LIN {X -117.977,Y -5.308,Z -33.189,A -90.000,B 90.000,C 0.000} C_DIS
LIN {X -117.973,Y -5.308,Z -33.170,A -90.000,B 90.000,C 0.000} C_DIS
LIN {X -117.912,Y -5.308,Z -32.912,A -90.000,B 90.000,C 0.000} C_DIS
LIN {X -117.911,Y -5.308,Z -32.907,A -90.000,B 90.000,C 0.000} C_DIS
LIN {X -117.908,Y -5.308,Z -32.898,A -90.000,B 90.000,C 0.000} C_DIS
LIN {X -117.792,Y -5.308,Z -32.451,A -90.000,B 90.000,C 0.000} C_DIS
LIN {X -117.766,Y -5.308,Z -32.368,A -90.000,B 90.000,C 0.000} C_DIS
LIN {X -117.707,Y -5.308,Z -32.184,A -90.000,B 90.000,C 0.000} C_DIS
LIN {X -117.545,Y -5.308,Z -31.754,A -90.000,B 90.000,C 0.000} C_DIS
LIN {X -117.540,Y -5.308,Z -31.738,A -90.000,B 90.000,C 0.000} C_DIS
LIN {X -117.536,Y -5.308,Z -31.729,A -90.000,B 90.000,C 0.000} C_DIS
LIN {X -117.439,Y -5.308,Z -31.478,A -90.000,B 90.000,C 0.000} C_DIS
LIN {X -117.430,Y -5.308,Z -31.458,A -90.000,B 90.000,C 0.000} C_DIS
LIN {X -117.326,Y -5.308,Z -31.223,A -90.000,B 90.000,C 0.000} C_DIS
LIN {X -117.220,Y -5.308,Z -31.001,A -90.000,B 90.000,C 0.000} C_DIS
LIN {X -117.148,Y -5.308,Z -30.851,A -90.000,B 90.000,C 0.000} C_DIS
LIN {X -117.070,Y -5.308,Z -30.695,A -90.000,B 90.000,C 0.000} C_DIS
LIN {X -117.022,Y -5.308,Z -30.598,A -90.000,B 90.000,C 0.000} C_DIS
LIN {X -116.974,Y -5.308,Z -30.507,A -90.000,B 90.000,C 0.000} C_DIS
LIN {X -116.886,Y -5.308,Z -30.345,A -90.000,B 90.000,C 0.000} C_DIS
LIN {X -116.807,Y -5.308,Z -30.208,A -90.000,B 90.000,C 0.000} C_DIS
LIN {X -116.654,Y -5.308,Z -29.940,A -90.000,B 90.000,C 0.000} C_DIS
LIN {X -116.605,Y -5.308,Z -29.858,A -90.000,B 90.000,C 0.000} C_DIS
LIN {X -116.503,Y -5.308,Z -29.690,A -90.000,B 90.000,C 0.000} C_DIS
LIN {X -116.452,Y -5.308,Z -29.616,A -90.000,B 90.000,C 0.000} C_DIS
LIN {X -116.331,Y -5.308,Z -29.445,A -90.000,B 90.000,C 0.000} C_DIS
LIN {X -116.254,Y -5.308,Z -29.338,A -90.000,B 90.000,C 0.000} C_DIS
LIN {X -116.057,Y -5.308,Z -29.066,A -90.000,B 90.000,C 0.000} C_DIS
LIN {X -116.003,Y -5.308,Z -29.001,A -90.000,B 90.000,C 0.000} C_DIS
LIN {X -115.858,Y -5.308,Z -28.827,A -90.000,B 90.000,C 0.000} C_DIS
LIN {X -115.778,Y -5.308,Z -28.738,A -90.000,B 90.000,C 0.000} C_DIS
LIN {X -115.545,Y -5.308,Z -28.480,A -90.000,B 90.000,C 0.000} C_DIS
LIN {X -115.368,Y -5.308,Z -28.303,A -90.000,B 90.000,C 0.000} C_DIS
LIN {X -115.313,Y -5.308,Z -28.248,A -90.000,B 90.000,C 0.000} C_DIS
LIN {X -115.111,Y -5.308,Z -28.056,A -90.000,B 90.000,C 0.000} C_DIS
LIN {X -115.057,Y -5.308,Z -28.004,A -90.000,B 90.000,C 0.000} C_DIS
LIN {X -114.997,Y -5.308,Z -27.943,A -90.000,B 90.000,C 0.000} C_DIS
LIN {X -114.943,Y -5.308,Z -27.887,A -90.000,B 90.000,C 0.000} C_DIS
LIN {X -114.922,Y -5.308,Z -27.862,A -90.000,B 90.000,C 0.000} C_DIS
LIN {X -114.912,Y -5.308,Z -27.851,A -90.000,B 90.000,C 0.000} C_DIS
LIN {X -114.867,Y -5.308,Z -27.784,A -90.000,B 90.000,C 0.000} C_DIS
LIN {X -114.827,Y -5.308,Z -27.724,A -90.000,B 90.000,C 0.000} C_DIS
LIN {X -114.791,Y -5.308,Z -27.667,A -90.000,B 90.000,C 0.000} C_DIS
LIN {X -114.554,Y -5.308,Z -27.272,A -90.000,B 90.000,C 0.000} C_DIS
LIN {X -114.525,Y -5.308,Z -27.224,A -90.000,B 90.000,C 0.000} C_DIS
LIN {X -114.272,Y -5.308,Z -26.790,A -90.000,B 90.000,C 0.000} C_DIS
LIN {X -114.249,Y -5.308,Z -26.755,A -90.000,B 90.000,C 0.000} C_DIS
LIN {X -113.974,Y -5.308,Z -26.300,A -90.000,B 90.000,C 0.000} C_DIS
LIN {X -113.958,Y -5.308,Z -26.278,A -90.000,B 90.000,C 0.000} C_DIS
LIN {X -113.653,Y -5.308,Z -25.822,A -90.000,B 90.000,C 0.000} C_DIS
LIN {X -113.650,Y -5.308,Z -25.818,A -90.000,B 90.000,C 0.000} C_DIS
LIN {X -113.644,Y -5.308,Z -25.810,A -90.000,B 90.000,C 0.000} C_DIS
LIN {X -113.382,Y -5.308,Z -25.448,A -90.000,B 90.000,C 0.000} C_DIS
LIN {X -113.086,Y -5.308,Z -25.058,A -90.000,B 90.000,C 0.000} C_DIS
LIN {X -113.033,Y -5.308,Z -24.989,A -90.000,B 90.000,C 0.000} C_DIS
LIN {X -113.032,Y -5.308,Z -24.987,A -90.000,B 90.000,C 0.000} C_DIS
LIN {X -112.663,Y -5.308,Z -24.567,A -90.000,B 90.000,C 0.000} C_DIS
LIN {X -112.656,Y -5.308,Z -24.559,A -90.000,B 90.000,C 0.000} C_DIS
LIN {X -112.516,Y -5.308,Z -24.404,A -90.000,B 90.000,C 0.000} C_DIS
LIN {X -112.449,Y -5.308,Z -24.329,A -90.000,B 90.000,C 0.000} C_DIS
LIN {X -112.346,Y -5.308,Z -24.216,A -90.000,B 90.000,C 0.000} C_DIS
LIN {X -112.343,Y -5.308,Z -24.212,A -90.000,B 90.000,C 0.000} C_DIS
LIN {X -111.943,Y -5.308,Z -23.828,A -90.000,B 90.000,C 0.000} C_DIS
LIN {X -111.933,Y -5.308,Z -23.819,A -90.000,B 90.000,C 0.000} C_DIS
LIN {X -111.792,Y -5.308,Z -23.682,A -90.000,B 90.000,C 0.000} C_DIS
LIN {X -111.722,Y -5.308,Z -23.614,A -90.000,B 90.000,C 0.000} C_DIS
LIN {X -111.540,Y -5.308,Z -23.467,A -90.000,B 90.000,C 0.000} C_DIS
LIN {X -111.368,Y -5.308,Z -23.328,A -90.000,B 90.000,C 0.000} C_DIS
LIN {X -111.135,Y -5.308,Z -23.144,A -90.000,B 90.000,C 0.000} C_DIS
LIN {X -110.924,Y -5.308,Z -22.980,A -90.000,B 90.000,C 0.000} C_DIS
LIN {X -110.660,Y -5.308,Z -22.810,A -90.000,B 90.000,C 0.000} C_DIS
LIN {X -110.453,Y -5.308,Z -22.678,A -90.000,B 90.000,C 0.000} C_DIS
LIN {X -110.276,Y -5.308,Z -22.565,A -90.000,B 90.000,C 0.000} C_DIS
LIN {X -110.054,Y -5.308,Z -22.425,A -90.000,B 90.000,C 0.000} C_DIS
LIN {X -109.741,Y -5.308,Z -22.262,A -90.000,B 90.000,C 0.000} C_DIS
LIN {X -109.517,Y -5.308,Z -22.148,A -90.000,B 90.000,C 0.000} C_DIS
LIN {X -109.275,Y -5.308,Z -22.028,A -90.000,B 90.000,C 0.000} C_DIS
LIN {X -109.109,Y -5.308,Z -21.946,A -90.000,B 90.000,C 0.000} C_DIS
LIN {X -108.725,Y -5.308,Z -21.782,A -90.000,B 90.000,C 0.000} C_DIS
LIN {X -108.517,Y -5.308,Z -21.696,A -90.000,B 90.000,C 0.000} C_DIS
LIN {X -108.363,Y -5.308,Z -21.637,A -90.000,B 90.000,C 0.000} C_DIS
LIN {X -108.231,Y -5.308,Z -21.589,A -90.000,B 90.000,C 0.000} C_DIS
LIN {X -107.827,Y -5.308,Z -21.447,A -90.000,B 90.000,C 0.000} C_DIS
LIN {X -107.525,Y -5.308,Z -21.341,A -90.000,B 90.000,C 0.000} C_DIS
LIN {X -107.463,Y -5.308,Z -21.320,A -90.000,B 90.000,C 0.000} C_DIS
LIN {X -107.432,Y -5.308,Z -21.310,A -90.000,B 90.000,C 0.000} C_DIS
LIN {X -107.310,Y -5.308,Z -21.274,A -90.000,B 90.000,C 0.000} C_DIS
LIN {X -107.063,Y -5.308,Z -21.202,A -90.000,B 90.000,C 0.000} C_DIS
LIN {X -106.666,Y -5.308,Z -21.088,A -90.000,B 90.000,C 0.000} C_DIS
LIN {X -106.324,Y -5.308,Z -21.004,A -90.000,B 90.000,C 0.000} C_DIS
LIN {X -106.187,Y -5.308,Z -20.973,A -90.000,B 90.000,C 0.000} C_DIS
LIN {X -105.726,Y -5.308,Z -20.868,A -90.000,B 90.000,C 0.000} C_DIS
LIN {X -105.570,Y -5.308,Z -20.834,A -90.000,B 90.000,C 0.000} C_DIS
LIN {X -105.545,Y -5.308,Z -20.829,A -90.000,B 90.000,C 0.000} C_DIS
LIN {X -104.926,Y -5.308,Z -20.730,A -90.000,B 90.000,C 0.000} C_DIS
LIN {X -104.782,Y -5.308,Z -20.706,A -90.000,B 90.000,C 0.000} C_DIS
LIN {X -104.613,Y -5.308,Z -20.683,A -90.000,B 90.000,C 0.000} C_DIS
LIN {X -104.426,Y -5.308,Z -20.658,A -90.000,B 90.000,C 0.000} C_DIS
LIN {X -104.379,Y -5.308,Z -20.652,A -90.000,B 90.000,C 0.000} C_DIS
LIN {X -104.331,Y -5.308,Z -20.646,A -90.000,B 90.000,C 0.000} C_DIS
LIN {X -104.108,Y -5.308,Z -20.623,A -90.000,B 90.000,C 0.000} C_DIS
LIN {X -103.651,Y -5.308,Z -20.576,A -90.000,B 90.000,C 0.000} C_DIS
LIN {X -103.189,Y -5.308,Z -20.536,A -90.000,B 90.000,C 0.000} C_DIS
LIN {X -102.818,Y -5.308,Z -20.508,A -90.000,B 90.000,C 0.000} C_DIS
LIN {X -102.806,Y -5.308,Z -20.507,A -90.000,B 90.000,C 0.000} C_DIS
LIN {X -102.635,Y -5.308,Z -20.494,A -90.000,B 90.000,C 0.000} C_DIS
LIN {X -102.599,Y -5.308,Z -20.490,A -90.000,B 90.000,C 0.000} C_DIS
LIN {X -102.490,Y -5.308,Z -20.481,A -90.000,B 90.000,C 0.000} C_DIS
LIN {X -102.372,Y -5.308,Z -20.470,A -90.000,B 90.000,C 0.000} C_DIS
LIN {X -102.183,Y -5.308,Z -20.453,A -90.000,B 90.000,C 0.000} C_DIS
LIN {X -102.123,Y -5.308,Z -20.445,A -90.000,B 90.000,C 0.000} C_DIS
LIN {X -101.878,Y -5.308,Z -20.411,A -90.000,B 90.000,C 0.000} C_DIS
LIN {X -101.864,Y -5.308,Z -20.409,A -90.000,B 90.000,C 0.000} C_DIS
LIN {X -101.846,Y -5.308,Z -20.405,A -90.000,B 90.000,C 0.000} C_DIS
LIN {X -101.761,Y -5.308,Z -20.383,A -90.000,B 90.000,C 0.000} C_DIS
LIN {X -101.660,Y -5.308,Z -20.356,A -90.000,B 90.000,C 0.000} C_DIS
LIN {X -101.653,Y -5.308,Z -20.354,A -90.000,B 90.000,C 0.000} C_DIS
LIN {X -101.547,Y -5.308,Z -20.319,A -90.000,B 90.000,C 0.000} C_DIS
LIN {X -101.451,Y -5.308,Z -20.286,A -90.000,B 90.000,C 0.000} C_DIS
LIN {X -101.435,Y -5.308,Z -20.280,A -90.000,B 90.000,C 0.000} C_DIS
LIN {X -101.428,Y -5.308,Z -20.278,A -90.000,B 90.000,C 0.000} C_DIS
LIN {X -101.398,Y -5.308,Z -20.264,A -90.000,B 90.000,C 0.000} C_DIS
LIN {X -101.267,Y -5.308,Z -20.207,A -90.000,B 90.000,C 0.000} C_DIS
LIN {X -101.212,Y -5.308,Z -20.183,A -90.000,B 90.000,C 0.000} C_DIS
LIN {X -101.176,Y -5.308,Z -20.167,A -90.000,B 90.000,C 0.000} C_DIS
LIN {X -101.175,Y -5.308,Z -20.167,A -90.000,B 90.000,C 0.000} C_DIS
LIN {X -101.139,Y -5.308,Z -20.148,A -90.000,B 90.000,C 0.000} C_DIS
LIN {X -101.032,Y -5.308,Z -20.093,A -90.000,B 90.000,C 0.000} C_DIS
LIN {X -100.951,Y -5.308,Z -20.051,A -90.000,B 90.000,C 0.000} C_DIS
LIN {X -100.946,Y -5.308,Z -20.048,A -90.000,B 90.000,C 0.000} C_DIS
LIN {X -100.942,Y -5.308,Z -20.046,A -90.000,B 90.000,C 0.000} C_DIS
LIN {X -100.936,Y -5.308,Z -20.042,A -90.000,B 90.000,C 0.000} C_DIS
LIN {X -100.934,Y -5.308,Z -20.041,A -90.000,B 90.000,C 0.000} C_DIS
LIN {X -100.933,Y -5.308,Z -20.040,A -90.000,B 90.000,C 0.000} C_DIS
LIN {X -100.930,Y -5.308,Z -20.038,A -90.000,B 90.000,C 0.000} C_DIS
LIN {X -100.928,Y -5.308,Z -20.036,A -90.000,B 90.000,C 0.000} C_DIS
LIN {X -100.849,Y -5.308,Z -19.968,A -90.000,B 90.000,C 0.000} C_DIS
LIN {X -100.827,Y -5.308,Z -19.949,A -90.000,B 90.000,C 0.000} C_DIS
LIN {X -100.826,Y -5.308,Z -19.948,A -90.000,B 90.000,C 0.000} C_DIS
LIN {X -100.790,Y -5.308,Z -19.914,A -90.000,B 90.000,C 0.000} C_DIS
LIN {X -100.739,Y -5.308,Z -19.865,A -90.000,B 90.000,C 0.000} C_DIS
LIN {X -100.635,Y -5.308,Z -19.765,A -90.000,B 90.000,C 0.000} C_DIS
LIN {X -100.472,Y -5.308,Z -19.608,A -90.000,B 90.000,C 0.000} C_DIS
LIN {X -100.461,Y -5.308,Z -19.597,A -90.000,B 90.000,C 0.000} C_DIS
LIN {X -100.415,Y -5.308,Z -19.556,A -90.000,B 90.000,C 0.000} C_DIS
LIN {X -100.383,Y -5.308,Z -19.526,A -90.000,B 90.000,C 0.000} C_DIS
LIN {X -100.369,Y -5.308,Z -19.513,A -90.000,B 90.000,C 0.000} C_DIS
LIN {X -100.363,Y -5.308,Z -19.508,A -90.000,B 90.000,C 0.000} C_DIS
LIN {X -100.186,Y -5.308,Z -19.343,A -90.000,B 90.000,C 0.000} C_DIS
LIN {X -100.167,Y -5.308,Z -19.325,A -90.000,B 90.000,C 0.000} C_DIS
LIN {X -100.162,Y -5.308,Z -19.321,A -90.000,B 90.000,C 0.000} C_DIS
LIN {X -100.071,Y -5.308,Z -19.246,A -90.000,B 90.000,C 0.000} C_DIS
LIN {X -100.050,Y -5.308,Z -19.227,A -90.000,B 90.000,C 0.000} C_DIS
LIN {X -100.032,Y -5.308,Z -19.212,A -90.000,B 90.000,C 0.000} C_DIS
LIN {X -99.996,Y -5.308,Z -19.182,A -90.000,B 90.000,C 0.000} C_DIS
LIN {X -99.990,Y -5.308,Z -19.176,A -90.000,B 90.000,C 0.000} C_DIS
LIN {X -99.909,Y -5.308,Z -19.108,A -90.000,B 90.000,C 0.000} C_DIS
LIN {X -99.832,Y -5.308,Z -19.043,A -90.000,B 90.000,C 0.000} C_DIS
LIN {X -99.763,Y -5.308,Z -18.987,A -90.000,B 90.000,C 0.000} C_DIS
LIN {X -99.751,Y -5.308,Z -18.977,A -90.000,B 90.000,C 0.000} C_DIS
LIN {X -99.628,Y -5.308,Z -18.878,A -90.000,B 90.000,C 0.000} C_DIS
LIN {X -99.614,Y -5.308,Z -18.867,A -90.000,B 90.000,C 0.000} C_DIS
LIN {X -99.597,Y -5.308,Z -18.853,A -90.000,B 90.000,C 0.000} C_DIS
LIN {X -99.494,Y -5.308,Z -18.770,A -90.000,B 90.000,C 0.000} C_DIS
LIN {X -99.478,Y -5.308,Z -18.757,A -90.000,B 90.000,C 0.000} C_DIS
LIN {X -99.449,Y -5.308,Z -18.736,A -90.000,B 90.000,C 0.000} C_DIS
LIN {X -99.433,Y -5.308,Z -18.724,A -90.000,B 90.000,C 0.000} C_DIS
LIN {X -99.382,Y -5.308,Z -18.686,A -90.000,B 90.000,C 0.000} C_DIS
LIN {X -99.381,Y -5.308,Z -18.686,A -90.000,B 90.000,C 0.000} C_DIS
LIN {X -99.381,Y -5.308,Z -18.685,A -90.000,B 90.000,C 0.000} C_DIS
LIN {X -99.378,Y -5.308,Z -18.684,A -90.000,B 90.000,C 0.000} C_DIS
LIN {X -99.378,Y -5.308,Z -18.683,A -90.000,B 90.000,C 0.000} C_DIS
LIN {X -99.303,Y -5.308,Z -18.628,A -90.000,B 90.000,C 0.000} C_DIS
LIN {X -99.176,Y -5.308,Z -18.534,A -90.000,B 90.000,C 0.000} C_DIS
LIN {X -99.109,Y -5.308,Z -18.483,A -90.000,B 90.000,C 0.000} C_DIS
LIN {X -99.100,Y -5.308,Z -18.477,A -90.000,B 90.000,C 0.000} C_DIS
LIN {X -98.932,Y -5.308,Z -18.363,A -90.000,B 90.000,C 0.000} C_DIS
LIN {X -98.923,Y -5.308,Z -18.356,A -90.000,B 90.000,C 0.000} C_DIS
LIN {X -98.845,Y -5.308,Z -18.303,A -90.000,B 90.000,C 0.000} C_DIS
LIN {X -98.780,Y -5.308,Z -18.259,A -90.000,B 90.000,C 0.000} C_DIS
LIN {X -98.724,Y -5.308,Z -18.220,A -90.000,B 90.000,C 0.000} C_DIS
LIN {X -98.646,Y -5.308,Z -18.167,A -90.000,B 90.000,C 0.000} C_DIS
LIN {X -98.634,Y -5.308,Z -18.159,A -90.000,B 90.000,C 0.000} C_DIS
LIN {X -98.620,Y -5.308,Z -18.149,A -90.000,B 90.000,C 0.000} C_DIS
LIN {X -98.612,Y -5.308,Z -18.144,A -90.000,B 90.000,C 0.000} C_DIS
LIN {X -98.598,Y -5.308,Z -18.134,A -90.000,B 90.000,C 0.000} C_DIS
LIN {X -98.583,Y -5.308,Z -18.124,A -90.000,B 90.000,C 0.000} C_DIS
LIN {X -98.579,Y -5.308,Z -18.122,A -90.000,B 90.000,C 0.000} C_DIS
LIN {X -98.572,Y -5.308,Z -18.118,A -90.000,B 90.000,C 0.000} C_DIS
LIN {X -98.562,Y -5.308,Z -18.113,A -90.000,B 90.000,C 0.000} C_DIS
LIN {X -98.534,Y -5.308,Z -18.097,A -90.000,B 90.000,C 0.000} C_DIS
LIN {X -98.379,Y -5.308,Z -17.995,A -90.000,B 90.000,C 0.000} C_DIS
LIN {X -98.319,Y -5.308,Z -17.960,A -90.000,B 90.000,C 0.000} C_DIS
LIN {X -98.088,Y -5.308,Z -17.826,A -90.000,B 90.000,C 0.000} C_DIS
LIN {X -98.049,Y -5.308,Z -17.804,A -90.000,B 90.000,C 0.000} C_DIS
LIN {X -97.929,Y -5.308,Z -17.727,A -90.000,B 90.000,C 0.000} C_DIS
LIN {X -97.896,Y -5.308,Z -17.706,A -90.000,B 90.000,C 0.000} C_DIS
LIN {X -97.858,Y -5.308,Z -17.682,A -90.000,B 90.000,C 0.000} C_DIS
LIN {X -97.794,Y -5.308,Z -17.642,A -90.000,B 90.000,C 0.000} C_DIS
LIN {X -97.770,Y -5.308,Z -17.626,A -90.000,B 90.000,C 0.000} C_DIS
LIN {X -97.761,Y -5.308,Z -17.621,A -90.000,B 90.000,C 0.000} C_DIS
LIN {X -97.650,Y -5.308,Z -17.564,A -90.000,B 90.000,C 0.000} C_DIS
LIN {X -97.617,Y -5.308,Z -17.548,A -90.000,B 90.000,C 0.000} C_DIS
LIN {X -97.579,Y -5.308,Z -17.528,A -90.000,B 90.000,C 0.000} C_DIS
LIN {X -97.512,Y -5.308,Z -17.493,A -90.000,B 90.000,C 0.000} C_DIS
LIN {X -97.347,Y -5.308,Z -17.408,A -90.000,B 90.000,C 0.000} C_DIS
LIN {X -97.177,Y -5.308,Z -17.329,A -90.000,B 90.000,C 0.000} C_DIS
LIN {X -97.111,Y -5.308,Z -17.296,A -90.000,B 90.000,C 0.000} C_DIS
LIN {X -96.869,Y -5.308,Z -17.173,A -90.000,B 90.000,C 0.000} C_DIS
LIN {X -96.730,Y -5.308,Z -17.106,A -90.000,B 90.000,C 0.000} C_DIS
LIN {X -96.682,Y -5.308,Z -17.083,A -90.000,B 90.000,C 0.000} C_DIS
LIN {X -96.630,Y -5.308,Z -17.058,A -90.000,B 90.000,C 0.000} C_DIS
LIN {X -96.621,Y -5.308,Z -17.054,A -90.000,B 90.000,C 0.000} C_DIS
LIN {X -96.612,Y -5.308,Z -17.049,A -90.000,B 90.000,C 0.000} C_DIS
LIN {X -96.448,Y -5.308,Z -16.970,A -90.000,B 90.000,C 0.000} C_DIS
LIN {X -96.434,Y -5.308,Z -16.964,A -90.000,B 90.000,C 0.000} C_DIS
LIN {X -96.428,Y -5.308,Z -16.962,A -90.000,B 90.000,C 0.000} C_DIS
LIN {X -96.231,Y -5.308,Z -16.890,A -90.000,B 90.000,C 0.000} C_DIS
LIN {X -96.223,Y -5.308,Z -16.886,A -90.000,B 90.000,C 0.000} C_DIS
LIN {X -96.020,Y -5.308,Z -16.809,A -90.000,B 90.000,C 0.000} C_DIS
LIN {X -95.841,Y -5.308,Z -16.740,A -90.000,B 90.000,C 0.000} C_DIS
LIN {X -95.569,Y -5.308,Z -16.634,A -90.000,B 90.000,C 0.000} C_DIS
LIN {X -95.454,Y -5.308,Z -16.588,A -90.000,B 90.000,C 0.000} C_DIS
LIN {X -95.323,Y -5.308,Z -16.544,A -90.000,B 90.000,C 0.000} C_DIS
LIN {X -95.275,Y -5.308,Z -16.527,A -90.000,B 90.000,C 0.000} C_DIS
LIN {X -95.094,Y -5.308,Z -16.465,A -90.000,B 90.000,C 0.000} C_DIS
LIN {X -94.993,Y -5.308,Z -16.431,A -90.000,B 90.000,C 0.000} C_DIS
LIN {X -94.698,Y -5.308,Z -16.347,A -90.000,B 90.000,C 0.000} C_DIS
LIN {X -94.682,Y -5.308,Z -16.342,A -90.000,B 90.000,C 0.000} C_DIS
LIN {X -94.588,Y -5.308,Z -16.315,A -90.000,B 90.000,C 0.000} C_DIS
LIN {X -94.583,Y -5.308,Z -16.313,A -90.000,B 90.000,C 0.000} C_DIS
LIN {X -94.569,Y -5.308,Z -16.307,A -90.000,B 90.000,C 0.000} C_DIS
LIN {X -94.419,Y -5.308,Z -16.245,A -90.000,B 90.000,C 0.000} C_DIS
LIN {X -94.350,Y -5.308,Z -16.215,A -90.000,B 90.000,C 0.000} C_DIS
LIN {X -94.183,Y -5.308,Z -16.142,A -90.000,B 90.000,C 0.000} C_DIS
LIN {X -94.163,Y -5.308,Z -16.134,A -90.000,B 90.000,C 0.000} C_DIS
LIN {X -93.756,Y -5.308,Z -15.976,A -90.000,B 90.000,C 0.000} C_DIS
LIN {X -93.754,Y -5.308,Z -15.976,A -90.000,B 90.000,C 0.000} C_DIS
LIN {X -93.686,Y -5.308,Z -15.949,A -90.000,B 90.000,C 0.000} C_DIS
LIN {X -93.246,Y -5.308,Z -15.767,A -90.000,B 90.000,C 0.000} C_DIS
LIN {X -93.175,Y -5.308,Z -15.738,A -90.000,B 90.000,C 0.000} C_DIS
LIN {X -93.133,Y -5.308,Z -15.722,A -90.000,B 90.000,C 0.000} C_DIS
LIN {X -93.130,Y -5.308,Z -15.721,A -90.000,B 90.000,C 0.000} C_DIS
LIN {X -92.911,Y -5.308,Z -15.642,A -90.000,B 90.000,C 0.000} C_DIS
LIN {X -92.907,Y -5.308,Z -15.641,A -90.000,B 90.000,C 0.000} C_DIS
LIN {X -92.118,Y -5.308,Z -15.333,A -90.000,B 90.000,C 0.000} C_DIS
LIN {X -92.116,Y -5.308,Z -15.332,A -90.000,B 90.000,C 0.000} C_DIS
LIN {X -92.077,Y -5.308,Z -15.318,A -90.000,B 90.000,C 0.000} C_DIS
LIN {X -91.313,Y -5.308,Z -15.046,A -90.000,B 90.000,C 0.000} C_DIS
LIN {X -90.936,Y -5.308,Z -14.907,A -90.000,B 90.000,C 0.000} C_DIS
LIN {X -90.928,Y -5.308,Z -14.904,A -90.000,B 90.000,C 0.000} C_DIS
LIN {X -90.891,Y -5.308,Z -14.890,A -90.000,B 90.000,C 0.000} C_DIS
LIN {X -90.585,Y -5.308,Z -14.790,A -90.000,B 90.000,C 0.000} C_DIS
LIN {X -89.802,Y -5.308,Z -14.535,A -90.000,B 90.000,C 0.000} C_DIS
LIN {X -89.667,Y -5.308,Z -14.493,A -90.000,B 90.000,C 0.000} C_DIS
LIN {X -88.942,Y -5.308,Z -14.279,A -90.000,B 90.000,C 0.000} C_DIS
LIN {X -88.377,Y -5.308,Z -14.113,A -90.000,B 90.000,C 0.000} C_DIS
LIN {X -88.302,Y -5.308,Z -14.092,A -90.000,B 90.000,C 0.000} C_DIS
LIN {X -87.613,Y -5.308,Z -13.901,A -90.000,B 90.000,C 0.000} C_DIS
LIN {X -87.198,Y -5.308,Z -13.791,A -90.000,B 90.000,C 0.000} C_DIS
LIN {X -87.088,Y -5.308,Z -13.765,A -90.000,B 90.000,C 0.000} C_DIS
LIN {X -86.190,Y -5.308,Z -13.541,A -90.000,B 90.000,C 0.000} C_DIS
LIN {X -85.658,Y -5.308,Z -13.422,A -90.000,B 90.000,C 0.000} C_DIS
LIN {X -84.346,Y -5.308,Z -13.105,A -90.000,B 90.000,C 0.000} C_DIS
LIN {X -84.206,Y -5.308,Z -13.073,A -90.000,B 90.000,C 0.000} C_DIS
LIN {X -84.188,Y -5.308,Z -13.070,A -90.000,B 90.000,C 0.000} C_DIS
LIN {X -84.122,Y -5.308,Z -13.056,A -90.000,B 90.000,C 0.000} C_DIS
LIN {X -82.940,Y -5.308,Z -12.809,A -90.000,B 90.000,C 0.000} C_DIS
LIN {X -82.725,Y -5.308,Z -12.767,A -90.000,B 90.000,C 0.000} C_DIS
LIN {X -81.589,Y -5.308,Z -12.563,A -90.000,B 90.000,C 0.000} C_DIS
LIN {X -81.273,Y -5.308,Z -12.506,A -90.000,B 90.000,C 0.000} C_DIS
LIN {X -81.158,Y -5.308,Z -12.488,A -90.000,B 90.000,C 0.000} C_DIS
LIN {X -80.762,Y -5.308,Z -12.437,A -90.000,B 90.000,C 0.000} C_DIS
LIN {X -79.898,Y -5.308,Z -12.335,A -90.000,B 90.000,C 0.000} C_DIS
LIN {X -79.532,Y -5.308,Z -12.302,A -90.000,B 90.000,C 0.000} C_DIS
LIN {X -79.431,Y -5.308,Z -12.297,A -90.000,B 90.000,C 0.000} C_DIS
LIN {X -79.069,Y -5.308,Z -12.279,A -90.000,B 90.000,C 0.000} C_DIS
LIN {X -78.172,Y -5.308,Z -12.237,A -90.000,B 90.000,C 0.000} C_DIS
LIN {X -77.499,Y -5.308,Z -12.247,A -90.000,B 90.000,C 0.000} C_DIS
LIN {X -77.013,Y -5.308,Z -12.254,A -90.000,B 90.000,C 0.000} C_DIS
LIN {X -76.853,Y -5.308,Z -12.258,A -90.000,B 90.000,C 0.000} C_DIS
LIN {X -76.541,Y -5.308,Z -12.273,A -90.000,B 90.000,C 0.000} C_DIS
LIN {X -76.282,Y -5.308,Z -12.288,A -90.000,B 90.000,C 0.000} C_DIS
LIN {X -76.107,Y -5.308,Z -12.298,A -90.000,B 90.000,C 0.000} C_DIS
LIN {X -75.514,Y -5.308,Z -12.340,A -90.000,B 90.000,C 0.000} C_DIS
LIN {X -75.035,Y -5.308,Z -12.381,A -90.000,B 90.000,C 0.000} C_DIS
LIN {X -74.511,Y -5.308,Z -12.438,A -90.000,B 90.000,C 0.000} C_DIS
LIN {X -74.265,Y -5.308,Z -12.469,A -90.000,B 90.000,C 0.000} C_DIS
LIN {X -74.047,Y -5.308,Z -12.497,A -90.000,B 90.000,C 0.000} C_DIS
LIN {X -73.867,Y -5.308,Z -12.520,A -90.000,B 90.000,C 0.000} C_DIS
LIN {X -73.549,Y -5.308,Z -12.555,A -90.000,B 90.000,C 0.000} C_DIS
LIN {X -73.267,Y -5.308,Z -12.590,A -90.000,B 90.000,C 0.000} C_DIS
LIN {X -73.086,Y -5.308,Z -12.613,A -90.000,B 90.000,C 0.000} C_DIS
LIN {X -73.010,Y -5.308,Z -12.624,A -90.000,B 90.000,C 0.000} C_DIS
LIN {X -72.780,Y -5.308,Z -12.656,A -90.000,B 90.000,C 0.000} C_DIS
LIN {X -72.699,Y -5.308,Z -12.666,A -90.000,B 90.000,C 0.000} C_DIS
LIN {X -72.236,Y -5.308,Z -12.719,A -90.000,B 90.000,C 0.000} C_DIS
LIN {X -72.223,Y -5.308,Z -12.721,A -90.000,B 90.000,C 0.000} C_DIS
LIN {X -72.209,Y -5.308,Z -12.723,A -90.000,B 90.000,C 0.000} C_DIS
LIN {X -72.158,Y -5.308,Z -12.729,A -90.000,B 90.000,C 0.000} C_DIS
LIN {X -71.257,Y -5.308,Z -12.826,A -90.000,B 90.000,C 0.000} C_DIS
LIN {X -71.170,Y -5.308,Z -12.836,A -90.000,B 90.000,C 0.000} C_DIS
LIN {X -71.139,Y -5.308,Z -12.839,A -90.000,B 90.000,C 0.000} C_DIS
LIN {X -71.133,Y -5.308,Z -12.840,A -90.000,B 90.000,C 0.000} C_DIS
LIN {X -71.130,Y -5.308,Z -12.840,A -90.000,B 90.000,C 0.000} C_DIS
LIN {X -70.477,Y -5.308,Z -12.894,A -90.000,B 90.000,C 0.000} C_DIS
LIN {X -69.402,Y -5.308,Z -12.947,A -90.000,B 90.000,C 0.000} C_DIS
LIN {X -69.331,Y -5.308,Z -12.950,A -90.000,B 90.000,C 0.000} C_DIS
LIN {X -69.304,Y -5.308,Z -12.952,A -90.000,B 90.000,C 0.000} C_DIS
LIN {X -69.167,Y -5.308,Z -12.961,A -90.000,B 90.000,C 0.000} C_DIS
LIN {X -67.794,Y -5.308,Z -13.016,A -90.000,B 90.000,C 0.000} C_DIS
LIN {X -67.759,Y -5.308,Z -13.018,A -90.000,B 90.000,C 0.000} C_DIS
LIN {X -67.483,Y -5.308,Z -13.032,A -90.000,B 90.000,C 0.000} C_DIS
LIN {X -66.325,Y -5.308,Z -13.101,A -90.000,B 90.000,C 0.000} C_DIS
LIN {X -65.936,Y -5.308,Z -13.135,A -90.000,B 90.000,C 0.000} C_DIS
LIN {X -65.714,Y -5.308,Z -13.157,A -90.000,B 90.000,C 0.000} C_DIS
LIN {X -64.626,Y -5.308,Z -13.260,A -90.000,B 90.000,C 0.000} C_DIS
LIN {X -64.483,Y -5.308,Z -13.279,A -90.000,B 90.000,C 0.000} C_DIS
LIN {X -64.039,Y -5.308,Z -13.351,A -90.000,B 90.000,C 0.000} C_DIS
LIN {X -63.215,Y -5.308,Z -13.484,A -90.000,B 90.000,C 0.000} C_DIS
LIN {X -62.959,Y -5.308,Z -13.536,A -90.000,B 90.000,C 0.000} C_DIS
LIN {X -62.424,Y -5.308,Z -13.650,A -90.000,B 90.000,C 0.000} C_DIS
LIN {X -61.835,Y -5.308,Z -13.776,A -90.000,B 90.000,C 0.000} C_DIS
LIN {X -61.594,Y -5.308,Z -13.833,A -90.000,B 90.000,C 0.000} C_DIS
LIN {X -60.935,Y -5.308,Z -13.995,A -90.000,B 90.000,C 0.000} C_DIS
LIN {X -60.497,Y -5.308,Z -14.102,A -90.000,B 90.000,C 0.000} C_DIS
LIN {X -59.682,Y -5.308,Z -14.305,A -90.000,B 90.000,C 0.000} C_DIS
LIN {X -59.680,Y -5.308,Z -14.305,A -90.000,B 90.000,C 0.000} C_DIS
LIN {X -59.664,Y -5.308,Z -14.309,A -90.000,B 90.000,C 0.000} C_DIS
LIN {X -59.164,Y -5.308,Z -14.419,A -90.000,B 90.000,C 0.000} C_DIS
LIN {X -59.057,Y -5.308,Z -14.443,A -90.000,B 90.000,C 0.000} C_DIS
LIN {X -58.999,Y -5.308,Z -14.457,A -90.000,B 90.000,C 0.000} C_DIS
LIN {X -58.894,Y -5.308,Z -14.481,A -90.000,B 90.000,C 0.000} C_DIS
LIN {X -58.803,Y -5.308,Z -14.502,A -90.000,B 90.000,C 0.000} C_DIS
LIN {X -57.871,Y -5.308,Z -14.708,A -90.000,B 90.000,C 0.000} C_DIS
LIN {X -57.379,Y -5.308,Z -14.819,A -90.000,B 90.000,C 0.000} C_DIS
LIN {X -56.779,Y -5.308,Z -14.954,A -90.000,B 90.000,C 0.000} C_DIS
LIN {X -56.593,Y -5.308,Z -14.998,A -90.000,B 90.000,C 0.000} C_DIS
LIN {X -55.769,Y -5.308,Z -15.194,A -90.000,B 90.000,C 0.000} C_DIS
LIN {X -55.466,Y -5.308,Z -15.267,A -90.000,B 90.000,C 0.000} C_DIS
LIN {X -54.314,Y -5.308,Z -15.565,A -90.000,B 90.000,C 0.000} C_DIS
LIN {X -54.115,Y -5.308,Z -15.617,A -90.000,B 90.000,C 0.000} C_DIS
LIN {X -53.717,Y -5.308,Z -15.722,A -90.000,B 90.000,C 0.000} C_DIS
LIN {X -52.558,Y -5.308,Z -16.029,A -90.000,B 90.000,C 0.000} C_DIS
LIN {X -52.458,Y -5.308,Z -16.055,A -90.000,B 90.000,C 0.000} C_DIS
LIN {X -51.843,Y -5.308,Z -16.216,A -90.000,B 90.000,C 0.000} C_DIS
LIN {X -51.840,Y -5.308,Z -16.217,A -90.000,B 90.000,C 0.000} C_DIS
LIN {X -51.696,Y -5.308,Z -16.255,A -90.000,B 90.000,C 0.000} C_DIS
LIN {X -51.415,Y -5.308,Z -16.329,A -90.000,B 90.000,C 0.000} C_DIS
LIN {X -51.382,Y -5.308,Z -16.338,A -90.000,B 90.000,C 0.000} C_DIS
LIN {X -50.449,Y -5.308,Z -16.585,A -90.000,B 90.000,C 0.000} C_DIS
LIN {X -50.377,Y -5.308,Z -16.603,A -90.000,B 90.000,C 0.000} C_DIS
LIN {X -50.372,Y -5.308,Z -16.604,A -90.000,B 90.000,C 0.000} C_DIS
LIN {X -50.349,Y -5.308,Z -16.609,A -90.000,B 90.000,C 0.000} C_DIS
LIN {X -47.942,Y -5.308,Z -17.229,A -90.000,B 90.000,C 0.000} C_DIS
LIN {X -47.364,Y -5.308,Z -17.356,A -90.000,B 90.000,C 0.000} C_DIS
LIN {X -44.859,Y -5.308,Z -17.966,A -90.000,B 90.000,C 0.000} C_DIS
LIN {X -43.325,Y -5.308,Z -18.281,A -90.000,B 90.000,C 0.000} C_DIS
LIN {X -42.883,Y -5.308,Z -18.373,A -90.000,B 90.000,C 0.000} C_DIS
LIN {X -42.882,Y -5.308,Z -18.373,A -90.000,B 90.000,C 0.000} C_DIS
LIN {X -42.876,Y -5.308,Z -18.375,A -90.000,B 90.000,C 0.000} C_DIS
LIN {X -42.211,Y -5.308,Z -18.513,A -90.000,B 90.000,C 0.000} C_DIS
LIN {X -41.586,Y -5.308,Z -18.658,A -90.000,B 90.000,C 0.000} C_DIS
LIN {X -39.389,Y -5.308,Z -19.089,A -90.000,B 90.000,C 0.000} C_DIS
LIN {X -38.060,Y -5.308,Z -19.353,A -90.000,B 90.000,C 0.000} C_DIS
LIN {X -37.751,Y -5.308,Z -19.407,A -90.000,B 90.000,C 0.000} C_DIS
LIN {X -34.672,Y -5.308,Z -20.017,A -90.000,B 90.000,C 0.000} C_DIS
LIN {X -33.753,Y -5.308,Z -20.192,A -90.000,B 90.000,C 0.000} C_DIS
LIN {X -31.674,Y -5.308,Z -20.626,A -90.000,B 90.000,C 0.000} C_DIS
LIN {X -30.395,Y -5.308,Z -20.891,A -90.000,B 90.000,C 0.000} C_DIS
LIN {X -29.981,Y -5.308,Z -20.978,A -90.000,B 90.000,C 0.000} C_DIS
LIN {X -29.405,Y -5.308,Z -21.098,A -90.000,B 90.000,C 0.000} C_DIS
LIN {X -28.688,Y -5.308,Z -21.256,A -90.000,B 90.000,C 0.000} C_DIS
LIN {X -26.533,Y -5.308,Z -21.733,A -90.000,B 90.000,C 0.000} C_DIS
LIN {X -26.208,Y -5.308,Z -21.807,A -90.000,B 90.000,C 0.000} C_DIS
LIN {X -23.880,Y -5.308,Z -22.341,A -90.000,B 90.000,C 0.000} C_DIS
LIN {X -23.861,Y -5.308,Z -22.346,A -90.000,B 90.000,C 0.000} C_DIS
LIN {X -23.846,Y -5.308,Z -22.349,A -90.000,B 90.000,C 0.000} C_DIS
LIN {X -23.703,Y -5.308,Z -22.382,A -90.000,B 90.000,C 0.000} C_DIS
LIN {X -21.692,Y -5.308,Z -22.852,A -90.000,B 90.000,C 0.000} C_DIS
LIN {X -19.797,Y -5.308,Z -23.300,A -90.000,B 90.000,C 0.000} C_DIS
LIN {X -19.515,Y -5.308,Z -23.367,A -90.000,B 90.000,C 0.000} C_DIS
LIN {X -19.091,Y -5.308,Z -23.468,A -90.000,B 90.000,C 0.000} C_DIS
LIN {X -18.785,Y -5.308,Z -23.541,A -90.000,B 90.000,C 0.000} C_DIS
LIN {X -16.916,Y -5.308,Z -23.995,A -90.000,B 90.000,C 0.000} C_DIS
LIN {X -16.673,Y -5.308,Z -24.054,A -90.000,B 90.000,C 0.000} C_DIS
LIN {X -14.686,Y -5.308,Z -24.546,A -90.000,B 90.000,C 0.000} C_DIS
LIN {X -14.099,Y -5.308,Z -24.694,A -90.000,B 90.000,C 0.000} C_DIS
LIN {X -13.235,Y -5.308,Z -24.920,A -90.000,B 90.000,C 0.000} C_DIS
LIN {X -11.276,Y -5.308,Z -25.420,A -90.000,B 90.000,C 0.000} C_DIS
LIN {X -9.754,Y -5.308,Z -25.819,A -90.000,B 90.000,C 0.000} C_DIS
LIN {X -8.276,Y -5.308,Z -26.195,A -90.000,B 90.000,C 0.000} C_DIS
LIN {X -6.013,Y -5.308,Z -26.767,A -90.000,B 90.000,C 0.000} C_DIS
LIN {X -5.335,Y -5.308,Z -26.933,A -90.000,B 90.000,C 0.000} C_DIS
LIN {X -5.322,Y -5.308,Z -26.936,A -90.000,B 90.000,C 0.000} C_DIS
LIN {X -2.602,Y -5.308,Z -27.572,A -90.000,B 90.000,C 0.000} C_DIS
LIN {X -2.596,Y -5.308,Z -27.573,A -90.000,B 90.000,C 0.000} C_DIS
LIN {X -2.506,Y -5.308,Z -27.594,A -90.000,B 90.000,C 0.000} C_DIS
LIN {X -2.444,Y -5.308,Z -27.606,A -90.000,B 90.000,C 0.000} C_DIS
LIN {X -2.142,Y -5.308,Z -27.668,A -90.000,B 90.000,C 0.000} C_DIS
LIN {X 0.618,Y -5.308,Z -28.236,A -90.000,B 90.000,C 0.000} C_DIS
LIN {X 1.331,Y -5.308,Z -28.369,A -90.000,B 90.000,C 0.000} C_DIS
LIN {X 3.580,Y -5.308,Z -28.826,A -90.000,B 90.000,C 0.000} C_DIS
LIN {X 4.649,Y -5.308,Z -29.035,A -90.000,B 90.000,C 0.000} C_DIS
LIN {X 6.298,Y -5.308,Z -29.381,A -90.000,B 90.000,C 0.000} C_DIS
LIN {X 6.751,Y -5.308,Z -29.473,A -90.000,B 90.000,C 0.000} C_DIS
LIN {X 8.715,Y -5.308,Z -29.892,A -90.000,B 90.000,C 0.000} C_DIS
LIN {X 9.672,Y -5.308,Z -30.095,A -90.000,B 90.000,C 0.000} C_DIS
LIN {X 10.782,Y -5.308,Z -30.356,A -90.000,B 90.000,C 0.000} C_DIS
LIN {X 12.055,Y -5.308,Z -30.626,A -90.000,B 90.000,C 0.000} C_DIS
LIN {X 12.170,Y -5.308,Z -30.654,A -90.000,B 90.000,C 0.000} C_DIS
LIN {X 12.485,Y -5.308,Z -30.730,A -90.000,B 90.000,C 0.000} C_DIS
LIN {X 13.426,Y -5.308,Z -30.925,A -90.000,B 90.000,C 0.000} C_DIS
LIN {X 14.187,Y -5.308,Z -31.082,A -90.000,B 90.000,C 0.000} C_DIS
LIN {X 14.730,Y -5.308,Z -31.191,A -90.000,B 90.000,C 0.000} C_DIS
LIN {X 15.822,Y -5.308,Z -31.428,A -90.000,B 90.000,C 0.000} C_DIS
LIN {X 16.879,Y -5.308,Z -31.640,A -90.000,B 90.000,C 0.000} C_DIS
LIN {X 17.496,Y -5.308,Z -31.763,A -90.000,B 90.000,C 0.000} C_DIS
LIN {X 18.119,Y -5.308,Z -31.880,A -90.000,B 90.000,C 0.000} C_DIS
LIN {X 18.131,Y -5.308,Z -31.882,A -90.000,B 90.000,C 0.000} C_DIS
LIN {X 18.348,Y -5.308,Z -31.923,A -90.000,B 90.000,C 0.000} C_DIS
LIN {X 19.045,Y -5.308,Z -32.062,A -90.000,B 90.000,C 0.000} C_DIS
LIN {X 19.171,Y -5.308,Z -32.087,A -90.000,B 90.000,C 0.000} C_DIS
LIN {X 19.575,Y -5.308,Z -32.164,A -90.000,B 90.000,C 0.000} C_DIS
LIN {X 19.702,Y -5.308,Z -32.188,A -90.000,B 90.000,C 0.000} C_DIS
LIN {X 20.520,Y -5.308,Z -32.344,A -90.000,B 90.000,C 0.000} C_DIS
LIN {X 21.907,Y -5.308,Z -32.600,A -90.000,B 90.000,C 0.000} C_DIS
LIN {X 21.908,Y -5.308,Z -32.600,A -90.000,B 90.000,C 0.000} C_DIS
LIN {X 22.387,Y -5.308,Z -32.691,A -90.000,B 90.000,C 0.000} C_DIS
LIN {X 22.389,Y -5.308,Z -32.692,A -90.000,B 90.000,C 0.000} C_DIS
LIN {X 23.854,Y -5.308,Z -32.973,A -90.000,B 90.000,C 0.000} C_DIS
LIN {X 23.856,Y -5.308,Z -32.974,A -90.000,B 90.000,C 0.000} C_DIS
LIN {X 23.913,Y -5.308,Z -32.985,A -90.000,B 90.000,C 0.000} C_DIS
LIN {X 25.280,Y -5.308,Z -33.266,A -90.000,B 90.000,C 0.000} C_DIS
LIN {X 25.285,Y -5.308,Z -33.267,A -90.000,B 90.000,C 0.000} C_DIS
LIN {X 25.403,Y -5.308,Z -33.294,A -90.000,B 90.000,C 0.000} C_DIS
LIN {X 26.733,Y -5.308,Z -33.598,A -90.000,B 90.000,C 0.000} C_DIS
LIN {X 26.742,Y -5.308,Z -33.600,A -90.000,B 90.000,C 0.000} C_DIS
LIN {X 26.951,Y -5.308,Z -33.654,A -90.000,B 90.000,C 0.000} C_DIS
LIN {X 28.279,Y -5.308,Z -33.999,A -90.000,B 90.000,C 0.000} C_DIS
LIN {X 28.291,Y -5.308,Z -34.003,A -90.000,B 90.000,C 0.000} C_DIS
LIN {X 28.317,Y -5.308,Z -34.010,A -90.000,B 90.000,C 0.000} C_DIS
LIN {X 28.345,Y -5.308,Z -34.019,A -90.000,B 90.000,C 0.000} C_DIS
LIN {X 29.634,Y -5.308,Z -34.397,A -90.000,B 90.000,C 0.000} C_DIS
LIN {X 29.981,Y -5.308,Z -34.499,A -90.000,B 90.000,C 0.000} C_DIS
LIN {X 29.985,Y -5.308,Z -34.500,A -90.000,B 90.000,C 0.000} C_DIS
LIN {X 30.049,Y -5.308,Z -34.519,A -90.000,B 90.000,C 0.000} C_DIS
LIN {X 30.073,Y -5.308,Z -34.527,A -90.000,B 90.000,C 0.000} C_DIS
LIN {X 30.402,Y -5.308,Z -34.625,A -90.000,B 90.000,C 0.000} C_DIS
LIN {X 30.448,Y -5.308,Z -34.638,A -90.000,B 90.000,C 0.000} C_DIS
LIN {X 30.467,Y -5.308,Z -34.644,A -90.000,B 90.000,C 0.000} C_DIS
LIN {X 30.515,Y -5.308,Z -34.660,A -90.000,B 90.000,C 0.000} C_DIS
LIN {X 30.946,Y -5.308,Z -34.797,A -90.000,B 90.000,C 0.000} C_DIS
LIN {X 32.183,Y -5.308,Z -35.190,A -90.000,B 90.000,C 0.000} C_DIS
LIN {X 32.240,Y -5.308,Z -35.208,A -90.000,B 90.000,C 0.000} C_DIS
LIN {X 32.311,Y -5.308,Z -35.231,A -90.000,B 90.000,C 0.000} C_DIS
LIN {X 32.337,Y -5.308,Z -35.239,A -90.000,B 90.000,C 0.000} C_DIS
LIN {X 32.358,Y -5.308,Z -35.247,A -90.000,B 90.000,C 0.000} C_DIS
LIN {X 32.613,Y -5.308,Z -35.332,A -90.000,B 90.000,C 0.000} C_DIS
LIN {X 33.589,Y -5.308,Z -35.659,A -90.000,B 90.000,C 0.000} C_DIS
LIN {X 33.980,Y -5.308,Z -35.790,A -90.000,B 90.000,C 0.000} C_DIS
LIN {X 34.129,Y -5.308,Z -35.836,A -90.000,B 90.000,C 0.000} C_DIS
LIN {X 34.326,Y -5.308,Z -35.898,A -90.000,B 90.000,C 0.000} C_DIS
LIN {X 34.347,Y -5.308,Z -35.905,A -90.000,B 90.000,C 0.000} C_DIS
LIN {X 34.381,Y -5.308,Z -35.916,A -90.000,B 90.000,C 0.000} C_DIS
LIN {X 34.591,Y -5.308,Z -35.983,A -90.000,B 90.000,C 0.000} C_DIS
LIN {X 35.286,Y -5.308,Z -36.206,A -90.000,B 90.000,C 0.000} C_DIS
LIN {X 35.555,Y -5.308,Z -36.292,A -90.000,B 90.000,C 0.000} C_DIS
LIN {X 36.507,Y -5.308,Z -36.597,A -90.000,B 90.000,C 0.000} C_DIS
LIN {X 36.549,Y -5.308,Z -36.610,A -90.000,B 90.000,C 0.000} C_DIS
LIN {X 36.619,Y -5.308,Z -36.633,A -90.000,B 90.000,C 0.000} C_DIS
LIN {X 38.006,Y -5.308,Z -37.081,A -90.000,B 90.000,C 0.000} C_DIS
LIN {X 38.926,Y -5.308,Z -37.378,A -90.000,B 90.000,C 0.000} C_DIS
LIN {X 38.963,Y -5.308,Z -37.390,A -90.000,B 90.000,C 0.000} C_DIS
LIN {X 39.047,Y -5.308,Z -37.418,A -90.000,B 90.000,C 0.000} C_DIS
LIN {X 39.290,Y -5.308,Z -37.501,A -90.000,B 90.000,C 0.000} C_DIS
LIN {X 39.464,Y -5.308,Z -37.560,A -90.000,B 90.000,C 0.000} C_DIS
LIN {X 40.739,Y -5.308,Z -37.941,A -90.000,B 90.000,C 0.000} C_DIS
LIN {X 41.425,Y -5.308,Z -38.147,A -90.000,B 90.000,C 0.000} C_DIS
LIN {X 41.554,Y -5.308,Z -38.190,A -90.000,B 90.000,C 0.000} C_DIS
LIN {X 41.699,Y -5.308,Z -38.238,A -90.000,B 90.000,C 0.000} C_DIS
LIN {X 41.945,Y -5.308,Z -38.320,A -90.000,B 90.000,C 0.000} C_DIS
LIN {X 42.270,Y -5.308,Z -38.428,A -90.000,B 90.000,C 0.000} C_DIS
LIN {X 42.411,Y -5.308,Z -38.475,A -90.000,B 90.000,C 0.000} C_DIS
LIN {X 42.646,Y -5.308,Z -38.553,A -90.000,B 90.000,C 0.000} C_DIS
LIN {X 43.221,Y -5.308,Z -38.720,A -90.000,B 90.000,C 0.000} C_DIS
LIN {X 43.430,Y -5.308,Z -38.780,A -90.000,B 90.000,C 0.000} C_DIS
LIN {X 43.460,Y -5.308,Z -38.789,A -90.000,B 90.000,C 0.000} C_DIS
LIN {X 43.719,Y -5.308,Z -38.866,A -90.000,B 90.000,C 0.000} C_DIS
LIN {X 43.793,Y -5.308,Z -38.888,A -90.000,B 90.000,C 0.000} C_DIS
LIN {X 43.897,Y -5.308,Z -38.920,A -90.000,B 90.000,C 0.000} C_DIS
LIN {X 44.075,Y -5.308,Z -38.982,A -90.000,B 90.000,C 0.000} C_DIS
LIN {X 45.081,Y -5.308,Z -39.335,A -90.000,B 90.000,C 0.000} C_DIS
LIN {X 45.917,Y -5.308,Z -39.629,A -90.000,B 90.000,C 0.000} C_DIS
LIN {X 46.496,Y -5.308,Z -39.833,A -90.000,B 90.000,C 0.000} C_DIS
LIN {X 46.609,Y -5.308,Z -39.873,A -90.000,B 90.000,C 0.000} C_DIS
LIN {X 46.940,Y -5.308,Z -40.010,A -90.000,B 90.000,C 0.000} C_DIS
LIN {X 47.027,Y -5.308,Z -40.046,A -90.000,B 90.000,C 0.000} C_DIS
LIN {X 47.060,Y -5.308,Z -40.059,A -90.000,B 90.000,C 0.000} C_DIS
LIN {X 47.238,Y -5.308,Z -40.136,A -90.000,B 90.000,C 0.000} C_DIS
LIN {X 47.876,Y -5.308,Z -40.414,A -90.000,B 90.000,C 0.000} C_DIS
LIN {X 48.771,Y -5.308,Z -40.804,A -90.000,B 90.000,C 0.000} C_DIS
LIN {X 49.152,Y -5.308,Z -40.969,A -90.000,B 90.000,C 0.000} C_DIS
LIN {X 49.312,Y -5.308,Z -41.039,A -90.000,B 90.000,C 0.000} C_DIS
LIN {X 49.484,Y -5.308,Z -41.114,A -90.000,B 90.000,C 0.000} C_DIS
LIN {X 49.505,Y -5.308,Z -41.124,A -90.000,B 90.000,C 0.000} C_DIS
LIN {X 49.527,Y -5.308,Z -41.136,A -90.000,B 90.000,C 0.000} C_DIS
LIN {X 49.687,Y -5.308,Z -41.217,A -90.000,B 90.000,C 0.000} C_DIS
LIN {X 49.716,Y -5.308,Z -41.231,A -90.000,B 90.000,C 0.000} C_DIS
LIN {X 49.904,Y -5.308,Z -41.332,A -90.000,B 90.000,C 0.000} C_DIS
LIN {X 50.265,Y -5.308,Z -41.523,A -90.000,B 90.000,C 0.000} C_DIS
LIN {X 50.265,Y -60.000,Z -41.523,A -90.000,B 90.000,C 0.000} C_DIS
LIN {X 103.582,Y -60.000,Z -88.349,A -90.000,B 90.000,C 0.000} C_DIS
LIN {X 103.582,Y -5.308,Z -88.349,A -90.000,B 90.000,C 0.000} C_DIS
LIN {X 103.597,Y -5.308,Z -88.382,A -90.000,B 90.000,C 0.000} C_DIS
LIN {X 104.150,Y -5.308,Z -89.512,A -90.000,B 90.000,C 0.000} C_DIS
LIN {X 104.260,Y -5.308,Z -89.777,A -90.000,B 90.000,C 0.000} C_DIS
LIN {X 104.694,Y -5.308,Z -90.775,A -90.000,B 90.000,C 0.000} C_DIS
LIN {X 104.828,Y -5.308,Z -91.132,A -90.000,B 90.000,C 0.000} C_DIS
LIN {X 104.865,Y -5.308,Z -91.230,A -90.000,B 90.000,C 0.000} C_DIS
LIN {X 105.198,Y -5.308,Z -92.121,A -90.000,B 90.000,C 0.000} C_DIS
LIN {X 105.286,Y -5.308,Z -92.369,A -90.000,B 90.000,C 0.000} C_DIS
LIN {X 105.556,Y -5.308,Z -93.223,A -90.000,B 90.000,C 0.000} C_DIS
LIN {X 105.622,Y -5.308,Z -93.442,A -90.000,B 90.000,C 0.000} C_DIS
LIN {X 105.860,Y -5.308,Z -94.318,A -90.000,B 90.000,C 0.000} C_DIS
LIN {X 105.961,Y -5.308,Z -94.703,A -90.000,B 90.000,C 0.000} C_DIS
LIN {X 105.984,Y -5.308,Z -94.789,A -90.000,B 90.000,C 0.000} C_DIS
LIN {X 106.034,Y -5.308,Z -94.984,A -90.000,B 90.000,C 0.000} C_DIS
LIN {X 106.272,Y -5.308,Z -95.943,A -90.000,B 90.000,C 0.000} C_DIS
LIN {X 106.312,Y -5.308,Z -96.113,A -90.000,B 90.000,C 0.000} C_DIS
LIN {X 106.583,Y -5.308,Z -97.223,A -90.000,B 90.000,C 0.000} C_DIS
LIN {X 106.617,Y -5.308,Z -97.360,A -90.000,B 90.000,C 0.000} C_DIS
LIN {X 106.931,Y -5.308,Z -98.677,A -90.000,B 90.000,C 0.000} C_DIS
LIN {X 106.954,Y -5.308,Z -98.771,A -90.000,B 90.000,C 0.000} C_DIS
LIN {X 107.321,Y -5.308,Z -100.347,A -90.000,B 90.000,C 0.000} C_DIS
LIN {X 107.331,Y -5.308,Z -100.389,A -90.000,B 90.000,C 0.000} C_DIS
LIN {X 107.691,Y -5.308,Z -101.975,A -90.000,B 90.000,C 0.000} C_DIS
LIN {X 107.748,Y -5.308,Z -102.228,A -90.000,B 90.000,C 0.000} C_DIS
LIN {X 107.755,Y -5.308,Z -102.261,A -90.000,B 90.000,C 0.000} C_DIS
LIN {X 108.198,Y -5.308,Z -104.269,A -90.000,B 90.000,C 0.000} C_DIS
LIN {X 108.234,Y -5.308,Z -104.434,A -90.000,B 90.000,C 0.000} C_DIS
LIN {X 108.696,Y -5.308,Z -106.615,A -90.000,B 90.000,C 0.000} C_DIS
LIN {X 108.747,Y -5.308,Z -106.856,A -90.000,B 90.000,C 0.000} C_DIS
LIN {X 109.210,Y -5.308,Z -109.189,A -90.000,B 90.000,C 0.000} C_DIS
LIN {X 109.266,Y -5.308,Z -109.474,A -90.000,B 90.000,C 0.000} C_DIS
LIN {X 109.702,Y -5.308,Z -111.878,A -90.000,B 90.000,C 0.000} C_DIS
LIN {X 109.767,Y -5.308,Z -112.237,A -90.000,B 90.000,C 0.000} C_DIS
LIN {X 110.139,Y -5.308,Z -114.561,A -90.000,B 90.000,C 0.000} C_DIS
LIN {X 110.225,Y -5.308,Z -115.095,A -90.000,B 90.000,C 0.000} C_DIS
LIN {X 110.240,Y -5.308,Z -115.190,A -90.000,B 90.000,C 0.000} C_DIS
LIN {X 110.299,Y -5.308,Z -115.575,A -90.000,B 90.000,C 0.000} C_DIS
LIN {X 110.599,Y -5.308,Z -117.677,A -90.000,B 90.000,C 0.000} C_DIS
LIN {X 110.711,Y -5.308,Z -118.466,A -90.000,B 90.000,C 0.000} C_DIS
LIN {X 110.937,Y -5.308,Z -120.242,A -90.000,B 90.000,C 0.000} C_DIS
LIN {X 111.075,Y -5.308,Z -121.332,A -90.000,B 90.000,C 0.000} C_DIS
LIN {X 111.232,Y -5.308,Z -122.713,A -90.000,B 90.000,C 0.000} C_DIS
LIN {X 111.391,Y -5.308,Z -124.110,A -90.000,B 90.000,C 0.000} C_DIS
LIN {X 111.488,Y -5.308,Z -125.070,A -90.000,B 90.000,C 0.000} C_DIS
LIN {X 111.656,Y -5.308,Z -126.742,A -90.000,B 90.000,C 0.000} C_DIS
LIN {X 111.702,Y -5.308,Z -127.297,A -90.000,B 90.000,C 0.000} C_DIS
LIN {X 111.705,Y -5.308,Z -127.324,A -90.000,B 90.000,C 0.000} C_DIS
LIN {X 111.870,Y -5.308,Z -129.316,A -90.000,B 90.000,C 0.000} C_DIS
LIN {X 111.872,Y -5.308,Z -129.337,A -90.000,B 90.000,C 0.000} C_DIS
LIN {X 111.958,Y -5.308,Z -130.723,A -90.000,B 90.000,C 0.000} C_DIS
LIN {X 112.020,Y -5.308,Z -131.781,A -90.000,B 90.000,C 0.000} C_DIS
LIN {X 112.031,Y -5.308,Z -131.973,A -90.000,B 90.000,C 0.000} C_DIS
LIN {X 112.033,Y -5.308,Z -132.014,A -90.000,B 90.000,C 0.000} C_DIS
LIN {X 112.056,Y -5.308,Z -132.455,A -90.000,B 90.000,C 0.000} C_DIS
LIN {X 112.136,Y -5.308,Z -134.612,A -90.000,B 90.000,C 0.000} C_DIS
LIN {X 112.160,Y -5.308,Z -135.256,A -90.000,B 90.000,C 0.000} C_DIS
LIN {X 112.192,Y -5.308,Z -137.123,A -90.000,B 90.000,C 0.000} C_DIS
LIN {X 112.213,Y -5.308,Z -138.317,A -90.000,B 90.000,C 0.000} C_DIS
LIN {X 112.214,Y -5.308,Z -139.796,A -90.000,B 90.000,C 0.000} C_DIS
LIN {X 112.215,Y -5.308,Z -141.602,A -90.000,B 90.000,C 0.000} C_DIS
LIN {X 112.200,Y -5.308,Z -142.623,A -90.000,B 90.000,C 0.000} C_DIS
LIN {X 112.164,Y -5.308,Z -145.075,A -90.000,B 90.000,C 0.000} C_DIS
LIN {X 112.162,Y -5.308,Z -145.197,A -90.000,B 90.000,C 0.000} C_DIS
LIN {X 112.161,Y -5.308,Z -145.226,A -90.000,B 90.000,C 0.000} C_DIS
LIN {X 112.062,Y -5.308,Z -148.699,A -90.000,B 90.000,C 0.000} C_DIS
LIN {X 112.054,Y -5.308,Z -148.896,A -90.000,B 90.000,C 0.000} C_DIS
LIN {X 111.917,Y -5.308,Z -152.041,A -90.000,B 90.000,C 0.000} C_DIS
LIN {X 111.898,Y -5.308,Z -152.483,A -90.000,B 90.000,C 0.000} C_DIS
LIN {X 111.882,Y -5.308,Z -152.838,A -90.000,B 90.000,C 0.000} C_DIS
LIN {X 111.722,Y -5.308,Z -155.799,A -90.000,B 90.000,C 0.000} C_DIS
LIN {X 111.676,Y -5.308,Z -156.654,A -90.000,B 90.000,C 0.000} C_DIS
LIN {X 111.510,Y -5.308,Z -159.303,A -90.000,B 90.000,C 0.000} C_DIS
LIN {X 111.433,Y -5.308,Z -160.526,A -90.000,B 90.000,C 0.000} C_DIS
LIN {X 111.268,Y -5.308,Z -162.894,A -90.000,B 90.000,C 0.000} C_DIS
LIN {X 111.161,Y -5.308,Z -164.425,A -90.000,B 90.000,C 0.000} C_DIS
LIN {X 111.001,Y -5.308,Z -166.546,A -90.000,B 90.000,C 0.000} C_DIS
LIN {X 110.868,Y -5.308,Z -168.319,A -90.000,B 90.000,C 0.000} C_DIS
LIN {X 110.713,Y -5.308,Z -170.207,A -90.000,B 90.000,C 0.000} C_DIS
LIN {X 110.557,Y -5.308,Z -172.121,A -90.000,B 90.000,C 0.000} C_DIS
LIN {X 110.407,Y -5.308,Z -173.802,A -90.000,B 90.000,C 0.000} C_DIS
LIN {X 110.234,Y -5.308,Z -175.744,A -90.000,B 90.000,C 0.000} C_DIS
LIN {X 110.209,Y -5.308,Z -176.025,A -90.000,B 90.000,C 0.000} C_DIS
LIN {X 110.203,Y -5.308,Z -176.093,A -90.000,B 90.000,C 0.000} C_DIS
LIN {X 109.908,Y -5.308,Z -179.082,A -90.000,B 90.000,C 0.000} C_DIS
LIN {X 109.876,Y -5.308,Z -179.406,A -90.000,B 90.000,C 0.000} C_DIS
LIN {X 109.579,Y -5.308,Z -182.082,A -90.000,B 90.000,C 0.000} C_DIS
LIN {X 109.544,Y -5.308,Z -182.383,A -90.000,B 90.000,C 0.000} C_DIS
LIN {X 109.247,Y -5.308,Z -184.805,A -90.000,B 90.000,C 0.000} C_DIS
LIN {X 109.211,Y -5.308,Z -185.093,A -90.000,B 90.000,C 0.000} C_DIS
LIN {X 109.157,Y -5.308,Z -185.503,A -90.000,B 90.000,C 0.000} C_DIS
LIN {X 109.150,Y -5.308,Z -185.556,A -90.000,B 90.000,C 0.000} C_DIS
LIN {X 108.905,Y -5.308,Z -187.401,A -90.000,B 90.000,C 0.000} C_DIS
LIN {X 108.871,Y -5.308,Z -187.656,A -90.000,B 90.000,C 0.000} C_DIS
LIN {X 108.823,Y -5.308,Z -188.019,A -90.000,B 90.000,C 0.000} C_DIS
LIN {X 108.816,Y -5.308,Z -188.073,A -90.000,B 90.000,C 0.000} C_DIS
LIN {X 108.519,Y -5.308,Z -190.203,A -90.000,B 90.000,C 0.000} C_DIS
LIN {X 108.483,Y -5.308,Z -190.473,A -90.000,B 90.000,C 0.000} C_DIS
LIN {X 108.184,Y -5.308,Z -192.578,A -90.000,B 90.000,C 0.000} C_DIS
LIN {X 108.147,Y -5.308,Z -192.847,A -90.000,B 90.000,C 0.000} C_DIS
LIN {X 107.808,Y -5.308,Z -195.145,A -90.000,B 90.000,C 0.000} C_DIS
LIN {X 107.769,Y -5.308,Z -195.410,A -90.000,B 90.000,C 0.000} C_DIS
LIN {X 107.349,Y -5.308,Z -198.131,A -90.000,B 90.000,C 0.000} C_DIS
LIN {X 107.312,Y -5.308,Z -198.368,A -90.000,B 90.000,C 0.000} C_DIS
LIN {X 106.768,Y -5.308,Z -201.761,A -90.000,B 90.000,C 0.000} C_DIS
LIN {X 106.106,Y -5.308,Z -205.755,A -90.000,B 90.000,C 0.000} C_DIS
LIN {X 106.036,Y -5.308,Z -206.182,A -90.000,B 90.000,C 0.000} C_DIS
LIN {X 106.024,Y -5.308,Z -206.254,A -90.000,B 90.000,C 0.000} C_DIS
LIN {X 105.265,Y -5.308,Z -210.470,A -90.000,B 90.000,C 0.000} C_DIS
LIN {X 105.108,Y -5.308,Z -211.343,A -90.000,B 90.000,C 0.000} C_DIS
LIN {X 105.091,Y -5.308,Z -211.434,A -90.000,B 90.000,C 0.000} C_DIS
LIN {X 104.335,Y -5.308,Z -215.184,A -90.000,B 90.000,C 0.000} C_DIS
LIN {X 103.968,Y -5.308,Z -217.008,A -90.000,B 90.000,C 0.000} C_DIS
LIN {X 103.272,Y -5.308,Z -220.015,A -90.000,B 90.000,C 0.000} C_DIS
LIN {X 102.640,Y -5.308,Z -222.750,A -90.000,B 90.000,C 0.000} C_DIS
LIN {X 102.591,Y -5.308,Z -222.951,A -90.000,B 90.000,C 0.000} C_DIS
LIN {X 101.995,Y -5.308,Z -225.136,A -90.000,B 90.000,C 0.000} C_DIS
LIN {X 101.060,Y -5.308,Z -228.562,A -90.000,B 90.000,C 0.000} C_DIS
LIN {X 100.587,Y -5.308,Z -230.086,A -90.000,B 90.000,C 0.000} C_DIS
LIN {X 99.299,Y -5.308,Z -234.243,A -90.000,B 90.000,C 0.000} C_DIS
LIN {X 99.186,Y -5.308,Z -234.605,A -90.000,B 90.000,C 0.000} C_DIS
LIN {X 98.898,Y -5.308,Z -235.454,A -90.000,B 90.000,C 0.000} C_DIS
LIN {X 97.213,Y -5.308,Z -240.417,A -90.000,B 90.000,C 0.000} C_DIS
LIN {X 97.167,Y -5.308,Z -240.554,A -90.000,B 90.000,C 0.000} C_DIS
LIN {X 97.164,Y -5.308,Z -240.561,A -90.000,B 90.000,C 0.000} C_DIS
LIN {X 96.078,Y -5.308,Z -243.561,A -90.000,B 90.000,C 0.000} C_DIS
LIN {X 96.078,Y -60.000,Z -243.561,A -90.000,B 90.000,C 0.000} C_DIS
LIN {X -120.015,Y -60.000,Z -236.852,A -90.000,B 90.000,C 0.000} C_DIS
LIN {X -120.015,Y -3.308,Z -236.852,A -90.000,B 90.000,C 0.000} C_DIS
LIN {X -119.372,Y -3.308,Z -236.429,A -90.000,B 90.000,C 0.000} C_DIS
LIN {X -115.376,Y -3.308,Z -233.808,A -90.000,B 90.000,C 0.000} C_DIS
LIN {X -111.910,Y -3.308,Z -231.538,A -90.000,B 90.000,C 0.000} C_DIS
LIN {X -106.958,Y -3.308,Z -228.330,A -90.000,B 90.000,C 0.000} C_DIS
LIN {X -104.157,Y -3.308,Z -226.519,A -90.000,B 90.000,C 0.000} C_DIS
LIN {X -98.145,Y -3.308,Z -222.710,A -90.000,B 90.000,C 0.000} C_DIS
LIN {X -96.125,Y -3.308,Z -221.431,A -90.000,B 90.000,C 0.000} C_DIS
LIN {X -96.034,Y -3.308,Z -221.375,A -90.000,B 90.000,C 0.000} C_DIS
LIN {X -95.714,Y -3.308,Z -221.178,A -90.000,B 90.000,C 0.000} C_DIS
LIN {X -88.418,Y -3.308,Z -216.700,A -90.000,B 90.000,C 0.000} C_DIS
LIN {X -87.413,Y -3.308,Z -216.083,A -90.000,B 90.000,C 0.000} C_DIS
LIN {X -86.652,Y -3.308,Z -215.633,A -90.000,B 90.000,C 0.000} C_DIS
LIN {X -81.125,Y -3.308,Z -212.384,A -90.000,B 90.000,C 0.000} C_DIS
LIN {X -78.834,Y -3.308,Z -211.043,A -90.000,B 90.000,C 0.000} C_DIS
LIN {X -73.527,Y -3.308,Z -208.009,A -90.000,B 90.000,C 0.000} C_DIS
LIN {X -70.331,Y -3.308,Z -206.183,A -90.000,B 90.000,C 0.000} C_DIS
LIN {X -69.089,Y -3.308,Z -205.478,A -90.000,B 90.000,C 0.000} C_DIS
LIN {X -63.160,Y -3.308,Z -202.126,A -90.000,B 90.000,C 0.000} C_DIS
LIN {X -62.367,Y -3.308,Z -201.680,A -90.000,B 90.000,C 0.000} C_DIS
LIN {X -56.746,Y -3.308,Z -198.459,A -90.000,B 90.000,C 0.000} C_DIS
LIN {X -56.671,Y -3.308,Z -198.416,A -90.000,B 90.000,C 0.000} C_DIS
LIN {X -55.393,Y -3.308,Z -197.688,A -90.000,B 90.000,C 0.000} C_DIS
LIN {X -51.410,Y -3.308,Z -195.298,A -90.000,B 90.000,C 0.000} C_DIS
LIN {X -49.931,Y -3.308,Z -194.415,A -90.000,B 90.000,C 0.000} C_DIS
LIN {X -46.547,Y -3.308,Z -192.273,A -90.000,B 90.000,C 0.000} C_DIS
LIN {X -45.167,Y -3.308,Z -191.402,A -90.000,B 90.000,C 0.000} C_DIS
LIN {X -42.383,Y -3.308,Z -189.537,A -90.000,B 90.000,C 0.000} C_DIS
LIN {X -41.173,Y -3.308,Z -188.728,A -90.000,B 90.000,C 0.000} C_DIS
LIN {X -38.742,Y -3.308,Z -187.014,A -90.000,B 90.000,C 0.000} C_DIS
LIN {X -37.691,Y -3.308,Z -186.274,A -90.000,B 90.000,C 0.000} C_DIS
LIN {X -36.801,Y -3.308,Z -185.626,A -90.000,B 90.000,C 0.000} C_DIS
LIN {X -36.730,Y -3.308,Z -185.574,A -90.000,B 90.000,C 0.000} C_DIS
LIN {X -34.715,Y -3.308,Z -184.104,A -90.000,B 90.000,C 0.000} C_DIS
LIN {X -34.713,Y -3.308,Z -184.102,A -90.000,B 90.000,C 0.000} C_DIS
LIN {X -34.712,Y -3.308,Z -184.101,A -90.000,B 90.000,C 0.000} C_DIS
LIN {X -34.010,Y -3.308,Z -183.566,A -90.000,B 90.000,C 0.000} C_DIS
LIN {X -33.910,Y -3.308,Z -183.490,A -90.000,B 90.000,C 0.000} C_DIS
LIN {X -31.907,Y -3.308,Z -181.960,A -90.000,B 90.000,C 0.000} C_DIS
LIN {X -31.181,Y -3.308,Z -181.372,A -90.000,B 90.000,C 0.000} C_DIS
LIN {X -29.246,Y -3.308,Z -179.801,A -90.000,B 90.000,C 0.000} C_DIS
LIN {X -28.644,Y -3.308,Z -179.272,A -90.000,B 90.000,C 0.000} C_DIS
LIN {X -27.123,Y -3.308,Z -177.933,A -90.000,B 90.000,C 0.000} C_DIS
LIN {X -25.704,Y -3.308,Z -176.546,A -90.000,B 90.000,C 0.000} C_DIS
LIN {X -25.684,Y -3.308,Z -176.526,A -90.000,B 90.000,C 0.000} C_DIS
LIN {X -25.654,Y -3.308,Z -176.497,A -90.000,B 90.000,C 0.000} C_DIS
LIN {X -25.218,Y -3.308,Z -176.071,A -90.000,B 90.000,C 0.000} C_DIS
LIN {X -24.070,Y -3.308,Z -174.788,A -90.000,B 90.000,C 0.000} C_DIS
LIN {X -23.825,Y -3.308,Z -174.515,A -90.000,B 90.000,C 0.000} C_DIS
LIN {X -23.766,Y -3.308,Z -174.449,A -90.000,B 90.000,C 0.000} C_DIS
LIN {X -22.654,Y -3.308,Z -173.000,A -90.000,B 90.000,C 0.000} C_DIS
LIN {X -22.511,Y -3.308,Z -172.815,A -90.000,B 90.000,C 0.000} C_DIS
LIN {X -22.511,Y -3.308,Z -172.814,A -90.000,B 90.000,C 0.000} C_DIS
LIN {X -22.402,Y -3.308,Z -172.671,A -90.000,B 90.000,C 0.000} C_DIS
LIN {X -22.398,Y -3.308,Z -172.665,A -90.000,B 90.000,C 0.000} C_DIS
LIN {X -21.352,Y -3.308,Z -171.061,A -90.000,B 90.000,C 0.000} C_DIS
LIN {X -21.316,Y -3.308,Z -171.006,A -90.000,B 90.000,C 0.000} C_DIS
LIN {X -21.305,Y -3.308,Z -170.988,A -90.000,B 90.000,C 0.000} C_DIS
LIN {X -21.151,Y -3.308,Z -170.751,A -90.000,B 90.000,C 0.000} C_DIS
LIN {X -21.150,Y -3.308,Z -170.749,A -90.000,B 90.000,C 0.000} C_DIS
LIN {X -20.171,Y -3.308,Z -168.990,A -90.000,B 90.000,C 0.000} C_DIS
LIN {X -20.151,Y -3.308,Z -168.954,A -90.000,B 90.000,C 0.000} C_DIS
LIN {X -20.151,Y -3.308,Z -168.953,A -90.000,B 90.000,C 0.000} C_DIS
LIN {X -20.026,Y -3.308,Z -168.727,A -90.000,B 90.000,C 0.000} C_DIS
LIN {X -19.051,Y -3.308,Z -166.689,A -90.000,B 90.000,C 0.000} C_DIS
LIN {X -19.000,Y -3.308,Z -166.582,A -90.000,B 90.000,C 0.000} C_DIS
LIN {X -18.249,Y -3.308,Z -164.706,A -90.000,B 90.000,C 0.000} C_DIS
LIN {X -18.191,Y -3.308,Z -164.561,A -90.000,B 90.000,C 0.000} C_DIS
LIN {X -18.190,Y -3.308,Z -164.559,A -90.000,B 90.000,C 0.000} C_DIS
LIN {X -18.133,Y -3.308,Z -164.374,A -90.000,B 90.000,C 0.000} C_DIS
LIN {X -18.063,Y -3.308,Z -164.147,A -90.000,B 90.000,C 0.000} C_DIS
LIN {X -17.963,Y -3.308,Z -163.824,A -90.000,B 90.000,C 0.000} C_DIS
LIN {X -17.755,Y -3.308,Z -163.150,A -90.000,B 90.000,C 0.000} C_DIS
LIN {X -17.728,Y -3.308,Z -163.064,A -90.000,B 90.000,C 0.000} C_DIS
LIN {X -17.586,Y -3.308,Z -162.186,A -90.000,B 90.000,C 0.000} C_DIS
LIN {X -17.583,Y -3.308,Z -162.171,A -90.000,B 90.000,C 0.000} C_DIS
LIN {X -17.582,Y -3.308,Z -162.161,A -90.000,B 90.000,C 0.000} C_DIS
LIN {X -17.583,Y -3.308,Z -162.125,A -90.000,B 90.000,C 0.000} C_DIS
LIN {X -17.593,Y -3.308,Z -161.737,A -90.000,B 90.000,C 0.000} C_DIS
LIN {X -17.593,Y -3.308,Z -161.708,A -90.000,B 90.000,C 0.000} C_DIS
LIN {X -17.679,Y -3.308,Z -161.321,A -90.000,B 90.000,C 0.000} C_DIS
LIN {X -17.685,Y -3.308,Z -161.294,A -90.000,B 90.000,C 0.000} C_DIS
LIN {X -17.894,Y -3.308,Z -160.722,A -90.000,B 90.000,C 0.000} C_DIS
LIN {X -17.996,Y -3.308,Z -160.445,A -90.000,B 90.000,C 0.000} C_DIS
LIN {X -18.364,Y -3.308,Z -159.553,A -90.000,B 90.000,C 0.000} C_DIS
LIN {X -18.364,Y -3.308,Z -159.552,A -90.000,B 90.000,C 0.000} C_DIS
LIN {X -18.378,Y -3.308,Z -159.525,A -90.000,B 90.000,C 0.000} C_DIS
LIN {X -18.402,Y -3.308,Z -159.480,A -90.000,B 90.000,C 0.000} C_DIS
LIN {X -18.486,Y -3.308,Z -159.322,A -90.000,B 90.000,C 0.000} C_DIS
LIN {X -18.517,Y -3.308,Z -159.264,A -90.000,B 90.000,C 0.000} C_DIS
LIN {X -18.524,Y -3.308,Z -159.251,A -90.000,B 90.000,C 0.000} C_DIS
LIN {X -18.909,Y -3.308,Z -158.523,A -90.000,B 90.000,C 0.000} C_DIS
LIN {X -18.960,Y -3.308,Z -158.451,A -90.000,B 90.000,C 0.000} C_DIS
LIN {X -18.962,Y -3.308,Z -158.447,A -90.000,B 90.000,C 0.000} C_DIS
LIN {X -18.999,Y -3.308,Z -158.392,A -90.000,B 90.000,C 0.000} C_DIS
LIN {X -19.002,Y -3.308,Z -158.388,A -90.000,B 90.000,C 0.000} C_DIS
LIN {X -19.826,Y -3.308,Z -157.168,A -90.000,B 90.000,C 0.000} C_DIS
LIN {X -19.950,Y -3.308,Z -157.020,A -90.000,B 90.000,C 0.000} C_DIS
LIN {X -19.988,Y -3.308,Z -156.973,A -90.000,B 90.000,C 0.000} C_DIS
LIN {X -19.992,Y -3.308,Z -156.968,A -90.000,B 90.000,C 0.000} C_DIS
LIN {X -21.349,Y -3.308,Z -155.303,A -90.000,B 90.000,C 0.000} C_DIS
LIN {X -21.496,Y -3.308,Z -155.148,A -90.000,B 90.000,C 0.000} C_DIS
LIN {X -21.614,Y -3.308,Z -155.022,A -90.000,B 90.000,C 0.000} C_DIS
LIN {X -23.727,Y -3.308,Z -152.761,A -90.000,B 90.000,C 0.000} C_DIS
LIN {X -24.047,Y -3.308,Z -152.425,A -90.000,B 90.000,C 0.000} C_DIS
LIN {X -26.668,Y -3.308,Z -149.636,A -90.000,B 90.000,C 0.000} C_DIS
LIN {X -26.998,Y -3.308,Z -149.264,A -90.000,B 90.000,C 0.000} C_DIS
LIN {X -29.761,Y -3.308,Z -146.108,A -90.000,B 90.000,C 0.000} C_DIS
LIN {X -29.795,Y -3.308,Z -146.069,A -90.000,B 90.000,C 0.000} C_DIS
LIN {X -30.079,Y -3.308,Z -145.740,A -90.000,B 90.000,C 0.000} C_DIS
LIN {X -30.397,Y -3.308,Z -145.328,A -90.000,B 90.000,C 0.000} C_DIS
LIN {X -33.036,Y -3.308,Z -141.861,A -90.000,B 90.000,C 0.000} C_DIS
LIN {X -33.067,Y -3.308,Z -141.816,A -90.000,B 90.000,C 0.000} C_DIS
LIN {X -33.314,Y -3.308,Z -141.462,A -90.000,B 90.000,C 0.000} C_DIS
LIN {X -33.611,Y -3.308,Z -140.977,A -90.000,B 90.000,C 0.000} C_DIS
LIN {X -35.845,Y -3.308,Z -137.287,A -90.000,B 90.000,C 0.000} C_DIS
LIN {X -35.848,Y -3.308,Z -137.281,A -90.000,B 90.000,C 0.000} C_DIS
LIN {X -35.866,Y -3.308,Z -137.251,A -90.000,B 90.000,C 0.000} C_DIS
LIN {X -35.924,Y -3.308,Z -137.146,A -90.000,B 90.000,C 0.000} C_DIS
LIN {X -36.080,Y -3.308,Z -136.861,A -90.000,B 90.000,C 0.000} C_DIS
LIN {X -36.089,Y -3.308,Z -136.844,A -90.000,B 90.000,C 0.000} C_DIS
LIN {X -36.089,Y -60.000,Z -136.844,A -90.000,B 90.000,C 0.000} C_DIS
LIN {X -44.232,Y -60.000,Z -119.970,A -90.000,B 90.000,C 0.000} C_DIS
LIN {X -44.232,Y -3.308,Z -119.970,A -90.000,B 90.000,C 0.000} C_DIS
LIN {X -44.277,Y -3.308,Z -119.907,A -90.000,B 90.000,C 0.000} C_DIS
LIN {X -44.386,Y -3.308,Z -119.751,A -90.000,B 90.000,C 0.000} C_DIS
LIN {X -44.856,Y -3.308,Z -119.088,A -90.000,B 90.000,C 0.000} C_DIS
LIN {X -45.653,Y -3.308,Z -118.051,A -90.000,B 90.000,C 0.000} C_DIS
LIN {X -46.328,Y -3.308,Z -117.172,A -90.000,B 90.000,C 0.000} C_DIS
LIN {X -47.244,Y -3.308,Z -116.024,A -90.000,B 90.000,C 0.000} C_DIS
LIN {X -48.100,Y -3.308,Z -114.953,A -90.000,B 90.000,C 0.000} C_DIS
LIN {X -49.070,Y -3.308,Z -113.753,A -90.000,B 90.000,C 0.000} C_DIS
LIN {X -50.114,Y -3.308,Z -112.472,A -90.000,B 90.000,C 0.000} C_DIS
LIN {X -51.100,Y -3.308,Z -111.247,A -90.000,B 90.000,C 0.000} C_DIS
LIN {X -52.316,Y -3.308,Z -109.763,A -90.000,B 90.000,C 0.000} C_DIS
LIN {X -52.491,Y -3.308,Z -109.542,A -90.000,B 90.000,C 0.000} C_DIS
LIN {X -52.527,Y -3.308,Z -109.496,A -90.000,B 90.000,C 0.000} C_DIS
LIN {X -52.798,Y -3.308,Z -109.154,A -90.000,B 90.000,C 0.000} C_DIS
LIN {X -54.511,Y -3.308,Z -107.047,A -90.000,B 90.000,C 0.000} C_DIS
LIN {X -54.524,Y -3.308,Z -107.031,A -90.000,B 90.000,C 0.000} C_DIS
LIN {X -54.564,Y -3.308,Z -106.982,A -90.000,B 90.000,C 0.000} C_DIS
LIN {X -54.798,Y -3.308,Z -106.689,A -90.000,B 90.000,C 0.000} C_DIS
LIN {X -56.996,Y -3.308,Z -104.024,A -90.000,B 90.000,C 0.000} C_DIS
LIN {X -57.108,Y -3.308,Z -103.888,A -90.000,B 90.000,C 0.000} C_DIS
LIN {X -57.942,Y -3.308,Z -102.914,A -90.000,B 90.000,C 0.000} C_DIS
LIN {X -58.372,Y -3.308,Z -102.411,A -90.000,B 90.000,C 0.000} C_DIS
LIN {X -58.871,Y -3.308,Z -101.829,A -90.000,B 90.000,C 0.000} C_DIS
LIN {X -59.295,Y -3.308,Z -101.350,A -90.000,B 90.000,C 0.000} C_DIS
LIN {X -61.013,Y -3.308,Z -99.466,A -90.000,B 90.000,C 0.000} C_DIS
LIN {X -61.030,Y -3.308,Z -99.448,A -90.000,B 90.000,C 0.000} C_DIS
LIN {X -61.072,Y -3.308,Z -99.401,A -90.000,B 90.000,C 0.000} C_DIS
LIN {X -61.094,Y -3.308,Z -99.378,A -90.000,B 90.000,C 0.000} C_DIS
LIN {X -61.435,Y -3.308,Z -99.013,A -90.000,B 90.000,C 0.000} C_DIS
LIN {X -61.449,Y -3.308,Z -98.999,A -90.000,B 90.000,C 0.000} C_DIS
LIN {X -63.382,Y -3.308,Z -97.089,A -90.000,B 90.000,C 0.000} C_DIS
LIN {X -63.580,Y -3.308,Z -96.894,A -90.000,B 90.000,C 0.000} C_DIS
LIN {X -63.594,Y -3.308,Z -96.881,A -90.000,B 90.000,C 0.000} C_DIS
LIN {X -64.583,Y -3.308,Z -96.002,A -90.000,B 90.000,C 0.000} C_DIS
LIN {X -65.896,Y -3.308,Z -94.829,A -90.000,B 90.000,C 0.000} C_DIS
LIN {X -66.785,Y -3.308,Z -94.117,A -90.000,B 90.000,C 0.000} C_DIS
LIN {X -66.940,Y -3.308,Z -93.993,A -90.000,B 90.000,C 0.000} C_DIS
LIN {X -67.916,Y -3.308,Z -93.203,A -90.000,B 90.000,C 0.000} C_DIS
LIN {X -67.935,Y -3.308,Z -93.189,A -90.000,B 90.000,C 0.000} C_DIS
LIN {X -68.052,Y -3.308,Z -93.103,A -90.000,B 90.000,C 0.000} C_DIS
LIN {X -68.729,Y -3.308,Z -92.610,A -90.000,B 90.000,C 0.000} C_DIS
LIN {X -68.766,Y -3.308,Z -92.583,A -90.000,B 90.000,C 0.000} C_DIS
LIN {X -69.768,Y -3.308,Z -91.841,A -90.000,B 90.000,C 0.000} C_DIS
LIN {X -69.942,Y -3.308,Z -91.713,A -90.000,B 90.000,C 0.000} C_DIS
LIN {X -70.075,Y -3.308,Z -91.615,A -90.000,B 90.000,C 0.000} C_DIS
LIN {X -70.078,Y -3.308,Z -91.612,A -90.000,B 90.000,C 0.000} C_DIS
LIN {X -70.695,Y -3.308,Z -91.196,A -90.000,B 90.000,C 0.000} C_DIS
LIN {X -70.698,Y -3.308,Z -91.194,A -90.000,B 90.000,C 0.000} C_DIS
LIN {X -71.108,Y -3.308,Z -90.917,A -90.000,B 90.000,C 0.000} C_DIS
LIN {X -71.534,Y -3.308,Z -90.628,A -90.000,B 90.000,C 0.000} C_DIS
LIN {X -72.184,Y -3.308,Z -90.188,A -90.000,B 90.000,C 0.000} C_DIS
LIN {X -73.248,Y -3.308,Z -89.504,A -90.000,B 90.000,C 0.000} C_DIS
LIN {X -74.339,Y -3.308,Z -88.807,A -90.000,B 90.000,C 0.000} C_DIS
LIN {X -74.466,Y -3.308,Z -88.727,A -90.000,B 90.000,C 0.000} C_DIS
LIN {X -76.022,Y -3.308,Z -87.756,A -90.000,B 90.000,C 0.000} C_DIS
LIN {X -76.167,Y -3.308,Z -87.665,A -90.000,B 90.000,C 0.000} C_DIS
LIN {X -76.347,Y -3.308,Z -87.553,A -90.000,B 90.000,C 0.000} C_DIS
LIN {X -76.371,Y -3.308,Z -87.537,A -90.000,B 90.000,C 0.000} C_DIS
LIN {X -76.576,Y -3.308,Z -87.406,A -90.000,B 90.000,C 0.000} C_DIS
LIN {X -77.821,Y -3.308,Z -86.608,A -90.000,B 90.000,C 0.000} C_DIS
LIN {X -78.192,Y -3.308,Z -86.372,A -90.000,B 90.000,C 0.000} C_DIS
LIN {X -79.180,Y -3.308,Z -85.688,A -90.000,B 90.000,C 0.000} C_DIS
LIN {X -79.760,Y -3.308,Z -85.285,A -90.000,B 90.000,C 0.000} C_DIS
LIN {X -79.989,Y -3.308,Z -85.121,A -90.000,B 90.000,C 0.000} C_DIS
LIN {X -80.153,Y -3.308,Z -85.004,A -90.000,B 90.000,C 0.000} C_DIS
LIN {X -80.867,Y -3.308,Z -84.476,A -90.000,B 90.000,C 0.000} C_DIS
LIN {X -81.508,Y -3.308,Z -83.999,A -90.000,B 90.000,C 0.000} C_DIS
LIN {X -82.081,Y -3.308,Z -83.556,A -90.000,B 90.000,C 0.000} C_DIS
LIN {X -82.703,Y -3.308,Z -83.075,A -90.000,B 90.000,C 0.000} C_DIS
LIN {X -83.211,Y -3.308,Z -82.676,A -90.000,B 90.000,C 0.000} C_DIS
LIN {X -83.792,Y -3.308,Z -82.228,A -90.000,B 90.000,C 0.000} C_DIS
LIN {X -83.900,Y -3.308,Z -82.146,A -90.000,B 90.000,C 0.000} C_DIS
LIN {X -83.990,Y -3.308,Z -82.077,A -90.000,B 90.000,C 0.000} C_DIS
LIN {X -83.994,Y -3.308,Z -82.074,A -90.000,B 90.000,C 0.000} C_DIS
LIN {X -84.568,Y -3.308,Z -81.656,A -90.000,B 90.000,C 0.000} C_DIS
LIN {X -84.573,Y -3.308,Z -81.652,A -90.000,B 90.000,C 0.000} C_DIS
LIN {X -85.545,Y -3.308,Z -80.975,A -90.000,B 90.000,C 0.000} C_DIS
LIN {X -85.551,Y -3.308,Z -80.971,A -90.000,B 90.000,C 0.000} C_DIS
LIN {X -86.460,Y -3.308,Z -80.353,A -90.000,B 90.000,C 0.000} C_DIS
LIN {X -86.469,Y -3.308,Z -80.346,A -90.000,B 90.000,C 0.000} C_DIS
LIN {X -87.262,Y -3.308,Z -79.806,A -90.000,B 90.000,C 0.000} C_DIS
LIN {X -87.308,Y -3.308,Z -79.774,A -90.000,B 90.000,C 0.000} C_DIS
LIN {X -87.996,Y -3.308,Z -79.288,A -90.000,B 90.000,C 0.000} C_DIS
LIN {X -88.084,Y -3.308,Z -79.225,A -90.000,B 90.000,C 0.000} C_DIS
LIN {X -88.670,Y -3.308,Z -78.807,A -90.000,B 90.000,C 0.000} C_DIS
LIN {X -88.795,Y -3.308,Z -78.717,A -90.000,B 90.000,C 0.000} C_DIS
LIN {X -88.841,Y -3.308,Z -78.686,A -90.000,B 90.000,C 0.000} C_DIS
LIN {X -88.848,Y -3.308,Z -78.681,A -90.000,B 90.000,C 0.000} C_DIS
LIN {X -88.855,Y -3.308,Z -78.676,A -90.000,B 90.000,C 0.000} C_DIS
LIN {X -88.868,Y -3.308,Z -78.667,A -90.000,B 90.000,C 0.000} C_DIS
LIN {X -89.415,Y -3.308,Z -78.284,A -90.000,B 90.000,C 0.000} C_DIS
LIN {X -89.497,Y -3.308,Z -78.232,A -90.000,B 90.000,C 0.000} C_DIS
LIN {X -89.501,Y -3.308,Z -78.229,A -90.000,B 90.000,C 0.000} C_DIS
LIN {X -89.513,Y -3.308,Z -78.221,A -90.000,B 90.000,C 0.000} C_DIS
LIN {X -89.662,Y -3.308,Z -78.123,A -90.000,B 90.000,C 0.000} C_DIS
LIN {X -89.723,Y -3.308,Z -78.083,A -90.000,B 90.000,C 0.000} C_DIS
LIN {X -89.724,Y -3.308,Z -78.083,A -90.000,B 90.000,C 0.000} C_DIS
LIN {X -89.811,Y -3.308,Z -78.032,A -90.000,B 90.000,C 0.000} C_DIS
LIN {X -90.028,Y -3.308,Z -77.906,A -90.000,B 90.000,C 0.000} C_DIS
LIN {X -90.032,Y -3.308,Z -77.904,A -90.000,B 90.000,C 0.000} C_DIS
LIN {X -90.035,Y -3.308,Z -77.903,A -90.000,B 90.000,C 0.000} C_DIS
LIN {X -90.071,Y -3.308,Z -77.887,A -90.000,B 90.000,C 0.000} C_DIS
LIN {X -90.072,Y -3.308,Z -77.887,A -90.000,B 90.000,C 0.000} C_DIS
LIN {X -90.277,Y -3.308,Z -77.885,A -90.000,B 90.000,C 0.000} C_DIS
LIN {X -90.295,Y -3.308,Z -77.885,A -90.000,B 90.000,C 0.000} C_DIS
LIN {X -90.510,Y -3.308,Z -77.884,A -90.000,B 90.000,C 0.000} C_DIS
LIN {X -91.247,Y -3.308,Z -77.924,A -90.000,B 90.000,C 0.000} C_DIS
LIN {X -91.384,Y -3.308,Z -77.928,A -90.000,B 90.000,C 0.000} C_DIS
LIN {X -91.430,Y -3.308,Z -77.930,A -90.000,B 90.000,C 0.000} C_DIS
LIN {X -92.154,Y -3.308,Z -77.962,A -90.000,B 90.000,C 0.000} C_DIS
LIN {X -92.457,Y -3.308,Z -77.979,A -90.000,B 90.000,C 0.000} C_DIS
LIN {X -93.013,Y -3.308,Z -77.993,A -90.000,B 90.000,C 0.000} C_DIS
LIN {X -93.605,Y -3.308,Z -78.024,A -90.000,B 90.000,C 0.000} C_DIS
LIN {X -93.948,Y -3.308,Z -78.017,A -90.000,B 90.000,C 0.000} C_DIS
LIN {X -93.989,Y -3.308,Z -78.016,A -90.000,B 90.000,C 0.000} C_DIS
LIN {X -94.071,Y -3.308,Z -78.018,A -90.000,B 90.000,C 0.000} C_DIS
LIN {X -94.904,Y -3.308,Z -78.034,A -90.000,B 90.000,C 0.000} C_DIS
LIN {X -95.139,Y -3.308,Z -78.025,A -90.000,B 90.000,C 0.000} C_DIS
LIN {X -95.357,Y -3.308,Z -78.014,A -90.000,B 90.000,C 0.000} C_DIS
LIN {X -95.412,Y -3.308,Z -78.009,A -90.000,B 90.000,C 0.000} C_DIS
LIN {X -96.316,Y -3.308,Z -77.951,A -90.000,B 90.000,C 0.000} C_DIS
LIN {X -96.768,Y -3.308,Z -77.922,A -90.000,B 90.000,C 0.000} C_DIS
LIN {X -97.128,Y -3.308,Z -77.869,A -90.000,B 90.000,C 0.000} C_DIS
LIN {X -97.237,Y -3.308,Z -77.851,A -90.000,B 90.000,C 0.000} C_DIS
LIN {X -98.553,Y -3.308,Z -77.605,A -90.000,B 90.000,C 0.000} C_DIS
LIN {X -98.737,Y -3.308,Z -77.571,A -90.000,B 90.000,C 0.000} C_DIS
LIN {X -98.785,Y -3.308,Z -77.562,A -90.000,B 90.000,C 0.000} C_DIS
LIN {X -98.803,Y -3.308,Z -77.558,A -90.000,B 90.000,C 0.000} C_DIS
LIN {X -99.149,Y -3.308,Z -77.465,A -90.000,B 90.000,C 0.000} C_DIS
LIN {X -99.197,Y -3.308,Z -77.452,A -90.000,B 90.000,C 0.000} C_DIS
LIN {X -99.238,Y -3.308,Z -77.438,A -90.000,B 90.000,C 0.000} C_DIS
LIN {X -99.253,Y -3.308,Z -77.433,A -90.000,B 90.000,C 0.000} C_DIS
LIN {X -100.315,Y -3.308,Z -77.068,A -90.000,B 90.000,C 0.000} C_DIS
LIN {X -100.855,Y -3.308,Z -76.895,A -90.000,B 90.000,C 0.000} C_DIS
LIN {X -101.149,Y -3.308,Z -76.778,A -90.000,B 90.000,C 0.000} C_DIS
LIN {X -101.289,Y -3.308,Z -76.722,A -90.000,B 90.000,C 0.000} C_DIS
LIN {X -101.568,Y -3.308,Z -76.574,A -90.000,B 90.000,C 0.000} C_DIS
LIN {X -101.702,Y -3.308,Z -76.504,A -90.000,B 90.000,C 0.000} C_DIS
LIN {X -102.181,Y -3.308,Z -76.246,A -90.000,B 90.000,C 0.000} C_DIS
LIN {X -102.898,Y -3.308,Z -75.862,A -90.000,B 90.000,C 0.000} C_DIS
LIN {X -103.325,Y -3.308,Z -75.633,A -90.000,B 90.000,C 0.000} C_DIS
LIN {X -103.352,Y -3.308,Z -75.619,A -90.000,B 90.000,C 0.000} C_DIS
LIN {X -103.361,Y -3.308,Z -75.614,A -90.000,B 90.000,C 0.000} C_DIS
LIN {X -103.606,Y -3.308,Z -75.455,A -90.000,B 90.000,C 0.000} C_DIS
LIN {X -103.723,Y -3.308,Z -75.376,A -90.000,B 90.000,C 0.000} C_DIS
LIN {X -104.623,Y -3.308,Z -74.759,A -90.000,B 90.000,C 0.000} C_DIS
LIN {X -105.376,Y -3.308,Z -74.243,A -90.000,B 90.000,C 0.000} C_DIS
LIN {X -105.532,Y -3.308,Z -74.120,A -90.000,B 90.000,C 0.000} C_DIS
LIN {X -105.979,Y -3.308,Z -73.755,A -90.000,B 90.000,C 0.000} C_DIS
LIN {X -106.968,Y -3.308,Z -72.950,A -90.000,B 90.000,C 0.000} C_DIS
LIN {X -107.269,Y -3.308,Z -72.700,A -90.000,B 90.000,C 0.000} C_DIS
LIN {X -108.063,Y -3.308,Z -71.952,A -90.000,B 90.000,C 0.000} C_DIS
LIN {X -108.637,Y -3.308,Z -71.426,A -90.000,B 90.000,C 0.000} C_DIS
LIN {X -108.804,Y -3.308,Z -71.261,A -90.000,B 90.000,C 0.000} C_DIS
LIN {X -108.977,Y -3.308,Z -71.092,A -90.000,B 90.000,C 0.000} C_DIS
LIN {X -109.615,Y -3.308,Z -70.406,A -90.000,B 90.000,C 0.000} C_DIS
LIN {X -110.085,Y -3.308,Z -69.894,A -90.000,B 90.000,C 0.000} C_DIS
LIN {X -110.275,Y -3.308,Z -69.664,A -90.000,B 90.000,C 0.000} C_DIS
LIN {X -110.388,Y -3.308,Z -69.527,A -90.000,B 90.000,C 0.000} C_DIS
LIN {X -111.042,Y -3.308,Z -68.662,A -90.000,B 90.000,C 0.000} C_DIS
LIN {X -111.297,Y -3.308,Z -68.322,A -90.000,B 90.000,C 0.000} C_DIS
LIN {X -111.494,Y -3.308,Z -68.024,A -90.000,B 90.000,C 0.000} C_DIS
LIN {X -111.560,Y -3.308,Z -67.925,A -90.000,B 90.000,C 0.000} C_DIS
LIN {X -112.210,Y -3.308,Z -66.831,A -90.000,B 90.000,C 0.000} C_DIS
LIN {X -112.329,Y -3.308,Z -66.631,A -90.000,B 90.000,C 0.000} C_DIS
LIN {X -112.375,Y -3.308,Z -66.545,A -90.000,B 90.000,C 0.000} C_DIS
LIN {X -112.528,Y -3.308,Z -66.252,A -90.000,B 90.000,C 0.000} C_DIS
LIN {X -112.542,Y -3.308,Z -66.222,A -90.000,B 90.000,C 0.000} C_DIS
LIN {X -112.549,Y -3.308,Z -66.208,A -90.000,B 90.000,C 0.000} C_DIS
LIN {X -113.206,Y -3.308,Z -64.813,A -90.000,B 90.000,C 0.000} C_DIS
LIN {X -113.238,Y -3.308,Z -64.746,A -90.000,B 90.000,C 0.000} C_DIS
LIN {X -113.249,Y -3.308,Z -64.721,A -90.000,B 90.000,C 0.000} C_DIS
LIN {X -113.408,Y -3.308,Z -64.317,A -90.000,B 90.000,C 0.000} C_DIS
LIN {X -113.460,Y -3.308,Z -64.185,A -90.000,B 90.000,C 0.000} C_DIS
LIN {X -113.756,Y -3.308,Z -63.427,A -90.000,B 90.000,C 0.000} C_DIS
LIN {X -114.019,Y -3.308,Z -62.745,A -90.000,B 90.000,C 0.000} C_DIS
LIN {X -114.066,Y -3.308,Z -62.622,A -90.000,B 90.000,C 0.000} C_DIS
LIN {X -114.080,Y -3.308,Z -62.583,A -90.000,B 90.000,C 0.000} C_DIS
LIN {X -114.598,Y -3.308,Z -61.096,A -90.000,B 90.000,C 0.000} C_DIS
LIN {X -114.735,Y -3.308,Z -60.701,A -90.000,B 90.000,C 0.000} C_DIS
LIN {X -115.165,Y -3.308,Z -59.423,A -90.000,B 90.000,C 0.000} C_DIS
LIN {X -115.388,Y -3.308,Z -58.757,A -90.000,B 90.000,C 0.000} C_DIS
LIN {X -115.729,Y -3.308,Z -57.768,A -90.000,B 90.000,C 0.000} C_DIS
LIN {X -115.975,Y -3.308,Z -57.052,A -90.000,B 90.000,C 0.000} C_DIS
LIN {X -116.187,Y -3.308,Z -56.485,A -90.000,B 90.000,C 0.000} C_DIS
LIN {X -116.203,Y -3.308,Z -56.444,A -90.000,B 90.000,C 0.000} C_DIS
LIN {X -116.592,Y -3.308,Z -55.405,A -90.000,B 90.000,C 0.000} C_DIS
LIN {X -116.701,Y -3.308,Z -55.116,A -90.000,B 90.000,C 0.000} C_DIS
LIN {X -116.924,Y -3.308,Z -54.527,A -90.000,B 90.000,C 0.000} C_DIS
LIN {X -117.254,Y -3.308,Z -53.680,A -90.000,B 90.000,C 0.000} C_DIS
LIN {X -117.405,Y -3.308,Z -53.239,A -90.000,B 90.000,C 0.000} C_DIS
LIN {X -117.739,Y -3.308,Z -52.298,A -90.000,B 90.000,C 0.000} C_DIS
LIN {X -117.838,Y -3.308,Z -51.941,A -90.000,B 90.000,C 0.000} C_DIS
LIN {X -117.866,Y -3.308,Z -51.839,A -90.000,B 90.000,C 0.000} C_DIS
LIN {X -117.930,Y -3.308,Z -51.589,A -90.000,B 90.000,C 0.000} C_DIS
LIN {X -118.182,Y -3.308,Z -50.631,A -90.000,B 90.000,C 0.000} C_DIS
LIN {X -118.211,Y -3.308,Z -50.462,A -90.000,B 90.000,C 0.000} C_DIS
LIN {X -118.236,Y -3.308,Z -50.315,A -90.000,B 90.000,C 0.000} C_DIS
LIN {X -118.252,Y -3.308,Z -50.214,A -90.000,B 90.000,C 0.000} C_DIS
LIN {X -118.260,Y -3.308,Z -50.161,A -90.000,B 90.000,C 0.000} C_DIS
LIN {X -118.278,Y -3.308,Z -49.996,A -90.000,B 90.000,C 0.000} C_DIS
LIN {X -118.293,Y -3.308,Z -49.851,A -90.000,B 90.000,C 0.000} C_DIS
LIN {X -118.356,Y -3.308,Z -49.080,A -90.000,B 90.000,C 0.000} C_DIS
LIN {X -118.381,Y -3.308,Z -48.795,A -90.000,B 90.000,C 0.000} C_DIS
LIN {X -118.383,Y -3.308,Z -48.657,A -90.000,B 90.000,C 0.000} C_DIS
LIN {X -118.388,Y -3.308,Z -48.328,A -90.000,B 90.000,C 0.000} C_DIS
LIN {X -118.346,Y -3.308,Z -47.707,A -90.000,B 90.000,C 0.000} C_DIS
LIN {X -118.327,Y -3.308,Z -47.422,A -90.000,B 90.000,C 0.000} C_DIS
LIN {X -118.312,Y -3.308,Z -47.265,A -90.000,B 90.000,C 0.000} C_DIS
LIN {X -118.284,Y -3.308,Z -46.957,A -90.000,B 90.000,C 0.000} C_DIS
LIN {X -118.202,Y -3.308,Z -46.454,A -90.000,B 90.000,C 0.000} C_DIS
LIN {X -118.156,Y -3.308,Z -46.173,A -90.000,B 90.000,C 0.000} C_DIS
LIN {X -118.090,Y -3.308,Z -45.775,A -90.000,B 90.000,C 0.000} C_DIS
LIN {X -118.083,Y -3.308,Z -45.735,A -90.000,B 90.000,C 0.000} C_DIS
LIN {X -118.083,Y -3.308,Z -45.732,A -90.000,B 90.000,C 0.000} C_DIS
LIN {X -118.084,Y -3.308,Z -45.723,A -90.000,B 90.000,C 0.000} C_DIS
LIN {X -118.085,Y -3.308,Z -45.710,A -90.000,B 90.000,C 0.000} C_DIS
LIN {X -118.085,Y -3.308,Z -45.709,A -90.000,B 90.000,C 0.000} C_DIS
LIN {X -118.085,Y -3.308,Z -45.708,A -90.000,B 90.000,C 0.000} C_DIS
LIN {X -118.111,Y -3.308,Z -45.598,A -90.000,B 90.000,C 0.000} C_DIS
LIN {X -118.116,Y -3.308,Z -45.581,A -90.000,B 90.000,C 0.000} C_DIS
LIN {X -118.119,Y -3.308,Z -45.571,A -90.000,B 90.000,C 0.000} C_DIS
LIN {X -118.123,Y -3.308,Z -45.559,A -90.000,B 90.000,C 0.000} C_DIS
LIN {X -118.141,Y -3.308,Z -45.498,A -90.000,B 90.000,C 0.000} C_DIS
LIN {X -118.154,Y -3.308,Z -45.456,A -90.000,B 90.000,C 0.000} C_DIS
LIN {X -118.244,Y -3.308,Z -45.162,A -90.000,B 90.000,C 0.000} C_DIS
LIN {X -118.297,Y -3.308,Z -44.975,A -90.000,B 90.000,C 0.000} C_DIS
LIN {X -118.384,Y -3.308,Z -44.672,A -90.000,B 90.000,C 0.000} C_DIS
LIN {X -118.454,Y -3.308,Z -44.428,A -90.000,B 90.000,C 0.000} C_DIS
LIN {X -118.513,Y -3.308,Z -44.216,A -90.000,B 90.000,C 0.000} C_DIS
LIN {X -118.554,Y -3.308,Z -44.052,A -90.000,B 90.000,C 0.000} C_DIS
LIN {X -118.580,Y -3.308,Z -43.951,A -90.000,B 90.000,C 0.000} C_DIS
LIN {X -118.667,Y -3.308,Z -43.588,A -90.000,B 90.000,C 0.000} C_DIS
LIN {X -118.706,Y -3.308,Z -43.413,A -90.000,B 90.000,C 0.000} C_DIS
LIN {X -118.767,Y -3.308,Z -43.052,A -90.000,B 90.000,C 0.000} C_DIS
LIN {X -118.821,Y -3.308,Z -42.728,A -90.000,B 90.000,C 0.000} C_DIS
LIN {X -118.845,Y -3.308,Z -42.582,A -90.000,B 90.000,C 0.000} C_DIS
LIN {X -118.870,Y -3.308,Z -42.420,A -90.000,B 90.000,C 0.000} C_DIS
LIN {X -118.893,Y -3.308,Z -42.061,A -90.000,B 90.000,C 0.000} C_DIS
LIN {X -118.913,Y -3.308,Z -41.721,A -90.000,B 90.000,C 0.000} C_DIS
LIN {X -118.921,Y -3.308,Z -41.585,A -90.000,B 90.000,C 0.000} C_DIS
LIN {X -118.928,Y -3.308,Z -41.443,A -90.000,B 90.000,C 0.000} C_DIS
LIN {X -118.913,Y -3.308,Z -41.100,A -90.000,B 90.000,C 0.000} C_DIS
LIN {X -118.907,Y -3.308,Z -40.967,A -90.000,B 90.000,C 0.000} C_DIS
LIN {X -118.890,Y -3.308,Z -40.612,A -90.000,B 90.000,C 0.000} C_DIS
LIN {X -118.883,Y -3.308,Z -40.494,A -90.000,B 90.000,C 0.000} C_DIS
LIN {X -118.863,Y -3.308,Z -40.317,A -90.000,B 90.000,C 0.000} C_DIS
LIN {X -118.840,Y -3.308,Z -40.120,A -90.000,B 90.000,C 0.000} C_DIS
LIN {X -118.829,Y -3.308,Z -40.050,A -90.000,B 90.000,C 0.000} C_DIS
LIN {X -118.762,Y -3.308,Z -39.684,A -90.000,B 90.000,C 0.000} C_DIS
LIN {X -118.745,Y -3.308,Z -39.600,A -90.000,B 90.000,C 0.000} C_DIS
LIN {X -118.670,Y -3.308,Z -39.226,A -90.000,B 90.000,C 0.000} C_DIS
LIN {X -118.646,Y -3.308,Z -39.152,A -90.000,B 90.000,C 0.000} C_DIS
LIN {X -118.620,Y -3.308,Z -39.068,A -90.000,B 90.000,C 0.000} C_DIS
LIN {X -118.506,Y -3.308,Z -38.707,A -90.000,B 90.000,C 0.000} C_DIS
LIN {X -118.400,Y -3.308,Z -38.385,A -90.000,B 90.000,C 0.000} C_DIS
LIN {X -118.361,Y -3.308,Z -38.297,A -90.000,B 90.000,C 0.000} C_DIS
LIN {X -118.212,Y -3.308,Z -37.957,A -90.000,B 90.000,C 0.000} C_DIS
LIN {X -118.068,Y -3.308,Z -37.676,A -90.000,B 90.000,C 0.000} C_DIS
LIN {X -118.032,Y -3.308,Z -37.606,A -90.000,B 90.000,C 0.000} C_DIS
LIN {X -118.018,Y -3.308,Z -37.582,A -90.000,B 90.000,C 0.000} C_DIS
LIN {X -118.000,Y -3.308,Z -37.550,A -90.000,B 90.000,C 0.000} C_DIS
LIN {X -117.984,Y -3.308,Z -37.522,A -90.000,B 90.000,C 0.000} C_DIS
LIN {X -117.977,Y -3.308,Z -37.510,A -90.000,B 90.000,C 0.000} C_DIS
LIN {X -117.978,Y -3.308,Z -37.507,A -90.000,B 90.000,C 0.000} C_DIS
LIN {X -118.052,Y -3.308,Z -37.273,A -90.000,B 90.000,C 0.000} C_DIS
LIN {X -118.073,Y -3.308,Z -37.206,A -90.000,B 90.000,C 0.000} C_DIS
LIN {X -118.076,Y -3.308,Z -37.197,A -90.000,B 90.000,C 0.000} C_DIS
LIN {X -118.086,Y -3.308,Z -37.166,A -90.000,B 90.000,C 0.000} C_DIS
LIN {X -118.205,Y -3.308,Z -36.777,A -90.000,B 90.000,C 0.000} C_DIS
LIN {X -118.288,Y -3.308,Z -36.508,A -90.000,B 90.000,C 0.000} C_DIS
LIN {X -118.314,Y -3.308,Z -36.397,A -90.000,B 90.000,C 0.000} C_DIS
LIN {X -118.368,Y -3.308,Z -36.173,A -90.000,B 90.000,C 0.000} C_DIS
LIN {X -118.395,Y -3.308,Z -36.038,A -90.000,B 90.000,C 0.000} C_DIS
LIN {X -118.463,Y -3.308,Z -35.695,A -90.000,B 90.000,C 0.000} C_DIS
LIN {X -118.474,Y -3.308,Z -35.620,A -90.000,B 90.000,C 0.000} C_DIS
LIN {X -118.506,Y -3.308,Z -35.397,A -90.000,B 90.000,C 0.000} C_DIS
LIN {X -118.514,Y -3.308,Z -35.318,A -90.000,B 90.000,C 0.000} C_DIS
LIN {X -118.529,Y -3.308,Z -35.170,A -90.000,B 90.000,C 0.000} C_DIS
LIN {X -118.557,Y -3.308,Z -34.869,A -90.000,B 90.000,C 0.000} C_DIS
LIN {X -118.564,Y -3.308,Z -34.679,A -90.000,B 90.000,C 0.000} C_DIS
LIN {X -118.567,Y -3.308,Z -34.603,A -90.000,B 90.000,C 0.000} C_DIS
LIN {X -118.569,Y -3.308,Z -34.484,A -90.000,B 90.000,C 0.000} C_DIS
LIN {X -118.569,Y -3.308,Z -34.214,A -90.000,B 90.000,C 0.000} C_DIS
LIN {X -118.569,Y -3.308,Z -34.069,A -90.000,B 90.000,C 0.000} C_DIS
LIN {X -118.560,Y -3.308,Z -33.914,A -90.000,B 90.000,C 0.000} C_DIS
LIN {X -118.553,Y -3.308,Z -33.790,A -90.000,B 90.000,C 0.000} C_DIS
LIN {X -118.531,Y -3.308,Z -33.533,A -90.000,B 90.000,C 0.000} C_DIS
LIN {X -118.512,Y -3.308,Z -33.309,A -90.000,B 90.000,C 0.000} C_DIS
LIN {X -118.494,Y -3.308,Z -33.169,A -90.000,B 90.000,C 0.000} C_DIS
LIN {X -118.475,Y -3.308,Z -33.030,A -90.000,B 90.000,C 0.000} C_DIS
LIN {X -118.431,Y -3.308,Z -32.802,A -90.000,B 90.000,C 0.000} C_DIS
LIN {X -118.383,Y -3.308,Z -32.556,A -90.000,B 90.000,C 0.000} C_DIS
LIN {X -118.358,Y -3.308,Z -32.430,A -90.000,B 90.000,C 0.000} C_DIS
LIN {X -118.326,Y -3.308,Z -32.279,A -90.000,B 90.000,C 0.000} C_DIS
LIN {X -118.295,Y -3.308,Z -32.168,A -90.000,B 90.000,C 0.000} C_DIS
LIN {X -118.250,Y -3.308,Z -32.008,A -90.000,B 90.000,C 0.000} C_DIS
LIN {X -118.196,Y -3.308,Z -31.829,A -90.000,B 90.000,C 0.000} C_DIS
LIN {X -118.110,Y -3.308,Z -31.546,A -90.000,B 90.000,C 0.000} C_DIS
LIN {X -118.051,Y -3.308,Z -31.378,A -90.000,B 90.000,C 0.000} C_DIS
LIN {X -118.018,Y -3.308,Z -31.282,A -90.000,B 90.000,C 0.000} C_DIS
LIN {X -117.980,Y -3.308,Z -31.183,A -90.000,B 90.000,C 0.000} C_DIS
LIN {X -117.904,Y -3.308,Z -30.987,A -90.000,B 90.000,C 0.000} C_DIS
LIN {X -117.846,Y -3.308,Z -30.849,A -90.000,B 90.000,C 0.000} C_DIS
LIN {X -117.810,Y -3.308,Z -30.763,A -90.000,B 90.000,C 0.000} C_DIS
LIN {X -117.737,Y -3.308,Z -30.590,A -90.000,B 90.000,C 0.000} C_DIS
LIN {X -117.688,Y -3.308,Z -30.489,A -90.000,B 90.000,C 0.000} C_DIS
LIN {X -117.615,Y -3.308,Z -30.336,A -90.000,B 90.000,C 0.000} C_DIS
LIN {X -117.495,Y -3.308,Z -30.096,A -90.000,B 90.000,C 0.000} C_DIS
LIN {X -117.440,Y -3.308,Z -29.991,A -90.000,B 90.000,C 0.000} C_DIS
LIN {X -117.375,Y -3.308,Z -29.868,A -90.000,B 90.000,C 0.000} C_DIS
LIN {X -117.261,Y -3.308,Z -29.660,A -90.000,B 90.000,C 0.000} C_DIS
LIN {X -117.188,Y -3.308,Z -29.529,A -90.000,B 90.000,C 0.000} C_DIS
LIN {X -117.120,Y -3.308,Z -29.409,A -90.000,B 90.000,C 0.000} C_DIS
LIN {X -117.031,Y -3.308,Z -29.266,A -90.000,B 90.000,C 0.000} C_DIS
LIN {X -116.964,Y -3.308,Z -29.160,A -90.000,B 90.000,C 0.000} C_DIS
LIN {X -116.860,Y -3.308,Z -28.998,A -90.000,B 90.000,C 0.000} C_DIS
LIN {X -116.697,Y -3.308,Z -28.762,A -90.000,B 90.000,C 0.000} C_DIS
LIN {X -116.586,Y -3.308,Z -28.608,A -90.000,B 90.000,C 0.000} C_DIS
LIN {X -116.520,Y -3.308,Z -28.516,A -90.000,B 90.000,C 0.000} C_DIS
LIN {X -116.414,Y -3.308,Z -28.383,A -90.000,B 90.000,C 0.000} C_DIS
LIN {X -116.286,Y -3.308,Z -28.231,A -90.000,B 90.000,C 0.000} C_DIS
LIN {X -116.224,Y -3.308,Z -28.158,A -90.000,B 90.000,C 0.000} C_DIS
LIN {X -116.008,Y -3.308,Z -27.905,A -90.000,B 90.000,C 0.000} C_DIS
LIN {X -115.904,Y -3.308,Z -27.800,A -90.000,B 90.000,C 0.000} C_DIS
LIN {X -115.744,Y -3.308,Z -27.639,A -90.000,B 90.000,C 0.000} C_DIS
LIN {X -115.683,Y -3.308,Z -27.578,A -90.000,B 90.000,C 0.000} C_DIS
LIN {X -115.500,Y -3.308,Z -27.394,A -90.000,B 90.000,C 0.000} C_DIS
LIN {X -115.487,Y -3.308,Z -27.381,A -90.000,B 90.000,C 0.000} C_DIS
LIN {X -115.456,Y -3.308,Z -27.347,A -90.000,B 90.000,C 0.000} C_DIS
LIN {X -115.452,Y -3.308,Z -27.342,A -90.000,B 90.000,C 0.000} C_DIS
LIN {X -115.442,Y -3.308,Z -27.331,A -90.000,B 90.000,C 0.000} C_DIS
LIN {X -115.398,Y -3.308,Z -27.284,A -90.000,B 90.000,C 0.000} C_DIS
LIN {X -115.317,Y -3.308,Z -27.199,A -90.000,B 90.000,C 0.000} C_DIS
LIN {X -115.314,Y -3.308,Z -27.196,A -90.000,B 90.000,C 0.000} C_DIS
LIN {X -115.312,Y -3.308,Z -27.193,A -90.000,B 90.000,C 0.000} C_DIS
LIN {X -115.310,Y -3.308,Z -27.191,A -90.000,B 90.000,C 0.000} C_DIS
LIN {X -115.300,Y -3.308,Z -27.175,A -90.000,B 90.000,C 0.000} C_DIS
LIN {X -115.296,Y -3.308,Z -27.167,A -90.000,B 90.000,C 0.000} C_DIS
LIN {X -115.280,Y -3.308,Z -27.140,A -90.000,B 90.000,C 0.000} C_DIS
LIN {X -115.165,Y -3.308,Z -26.942,A -90.000,B 90.000,C 0.000} C_DIS
LIN {X -115.037,Y -3.308,Z -26.708,A -90.000,B 90.000,C 0.000} C_DIS
LIN {X -114.906,Y -3.308,Z -26.476,A -90.000,B 90.000,C 0.000} C_DIS
LIN {X -114.768,Y -3.308,Z -26.214,A -90.000,B 90.000,C 0.000} C_DIS
LIN {X -114.639,Y -3.308,Z -25.994,A -90.000,B 90.000,C 0.000} C_DIS
LIN {X -114.485,Y -3.308,Z -25.714,A -90.000,B 90.000,C 0.000} C_DIS
LIN {X -114.375,Y -3.308,Z -25.543,A -90.000,B 90.000,C 0.000} C_DIS
LIN {X -114.326,Y -3.308,Z -25.466,A -90.000,B 90.000,C 0.000} C_DIS
LIN {X -114.211,Y -3.308,Z -25.280,A -90.000,B 90.000,C 0.000} C_DIS
LIN {X -114.181,Y -3.308,Z -25.232,A -90.000,B 90.000,C 0.000} C_DIS
LIN {X -114.080,Y -3.308,Z -25.074,A -90.000,B 90.000,C 0.000} C_DIS
LIN {X -113.924,Y -3.308,Z -24.831,A -90.000,B 90.000,C 0.000} C_DIS
LIN {X -113.796,Y -3.308,Z -24.656,A -90.000,B 90.000,C 0.000} C_DIS
LIN {X -113.595,Y -3.308,Z -24.373,A -90.000,B 90.000,C 0.000} C_DIS
LIN {X -113.541,Y -3.308,Z -24.304,A -90.000,B 90.000,C 0.000} C_DIS
LIN {X -113.432,Y -3.308,Z -24.163,A -90.000,B 90.000,C 0.000} C_DIS
LIN {X -113.354,Y -3.308,Z -24.066,A -90.000,B 90.000,C 0.000} C_DIS
LIN {X -113.255,Y -3.308,Z -23.948,A -90.000,B 90.000,C 0.000} C_DIS
LIN {X -112.994,Y -3.308,Z -23.636,A -90.000,B 90.000,C 0.000} C_DIS
LIN {X -112.779,Y -3.308,Z -23.398,A -90.000,B 90.000,C 0.000} C_DIS
LIN {X -112.674,Y -3.308,Z -23.292,A -90.000,B 90.000,C 0.000} C_DIS
LIN {X -112.546,Y -3.308,Z -23.167,A -90.000,B 90.000,C 0.000} C_DIS
LIN {X -112.278,Y -3.308,Z -22.904,A -90.000,B 90.000,C 0.000} C_DIS
LIN {X -112.050,Y -3.308,Z -22.700,A -90.000,B 90.000,C 0.000} C_DIS
LIN {X -111.923,Y -3.308,Z -22.596,A -90.000,B 90.000,C 0.000} C_DIS
LIN {X -111.771,Y -3.308,Z -22.477,A -90.000,B 90.000,C 0.000} C_DIS
LIN {X -111.488,Y -3.308,Z -22.257,A -90.000,B 90.000,C 0.000} C_DIS
LIN {X -111.243,Y -3.308,Z -22.081,A -90.000,B 90.000,C 0.000} C_DIS
LIN {X -111.102,Y -3.308,Z -21.988,A -90.000,B 90.000,C 0.000} C_DIS
LIN {X -110.935,Y -3.308,Z -21.884,A -90.000,B 90.000,C 0.000} C_DIS
LIN {X -110.627,Y -3.308,Z -21.692,A -90.000,B 90.000,C 0.000} C_DIS
LIN {X -110.360,Y -3.308,Z -21.540,A -90.000,B 90.000,C 0.000} C_DIS
LIN {X -110.215,Y -3.308,Z -21.466,A -90.000,B 90.000,C 0.000} C_DIS
LIN {X -110.045,Y -3.308,Z -21.380,A -90.000,B 90.000,C 0.000} C_DIS
LIN {X -109.701,Y -3.308,Z -21.205,A -90.000,B 90.000,C 0.000} C_DIS
LIN {X -109.402,Y -3.308,Z -21.076,A -90.000,B 90.000,C 0.000} C_DIS
LIN {X -109.236,Y -3.308,Z -21.006,A -90.000,B 90.000,C 0.000} C_DIS
LIN {X -108.819,Y -3.308,Z -20.833,A -90.000,B 90.000,C 0.000} C_DIS
LIN {X -108.712,Y -3.308,Z -20.792,A -90.000,B 90.000,C 0.000} C_DIS
LIN {X -108.582,Y -3.308,Z -20.746,A -90.000,B 90.000,C 0.000} C_DIS
LIN {X -108.115,Y -3.308,Z -20.583,A -90.000,B 90.000,C 0.000} C_DIS
LIN {X -107.734,Y -3.308,Z -20.465,A -90.000,B 90.000,C 0.000} C_DIS
LIN {X -107.645,Y -3.308,Z -20.439,A -90.000,B 90.000,C 0.000} C_DIS
LIN {X -107.056,Y -3.308,Z -20.267,A -90.000,B 90.000,C 0.000} C_DIS
LIN {X -107.043,Y -3.308,Z -20.264,A -90.000,B 90.000,C 0.000} C_DIS
LIN {X -107.027,Y -3.308,Z -20.260,A -90.000,B 90.000,C 0.000} C_DIS
LIN {X -106.916,Y -3.308,Z -20.233,A -90.000,B 90.000,C 0.000} C_DIS
LIN {X -106.420,Y -3.308,Z -20.115,A -90.000,B 90.000,C 0.000} C_DIS
LIN {X -106.378,Y -3.308,Z -20.105,A -90.000,B 90.000,C 0.000} C_DIS
LIN {X -106.336,Y -3.308,Z -20.096,A -90.000,B 90.000,C 0.000} C_DIS
LIN {X -106.124,Y -3.308,Z -20.050,A -90.000,B 90.000,C 0.000} C_DIS
LIN {X -105.912,Y -3.308,Z -20.010,A -90.000,B 90.000,C 0.000} C_DIS
LIN {X -105.425,Y -3.308,Z -19.920,A -90.000,B 90.000,C 0.000} C_DIS
LIN {X -105.334,Y -3.308,Z -19.904,A -90.000,B 90.000,C 0.000} C_DIS
LIN {X -105.238,Y -3.308,Z -19.887,A -90.000,B 90.000,C 0.000} C_DIS
LIN {X -105.112,Y -3.308,Z -19.868,A -90.000,B 90.000,C 0.000} C_DIS
LIN {X -104.955,Y -3.308,Z -19.843,A -90.000,B 90.000,C 0.000} C_DIS
LIN {X -104.303,Y -3.308,Z -19.761,A -90.000,B 90.000,C 0.000} C_DIS
LIN {X -104.261,Y -3.308,Z -19.755,A -90.000,B 90.000,C 0.000} C_DIS
LIN {X -104.044,Y -3.308,Z -19.733,A -90.000,B 90.000,C 0.000} C_DIS
LIN {X -103.722,Y -3.308,Z -19.702,A -90.000,B 90.000,C 0.000} C_DIS
LIN {X -103.633,Y -3.308,Z -19.694,A -90.000,B 90.000,C 0.000} C_DIS
LIN {X -103.439,Y -3.308,Z -19.672,A -90.000,B 90.000,C 0.000} C_DIS
LIN {X -103.395,Y -3.308,Z -19.667,A -90.000,B 90.000,C 0.000} C_DIS
LIN {X -103.344,Y -3.308,Z -19.660,A -90.000,B 90.000,C 0.000} C_DIS
LIN {X -103.233,Y -3.308,Z -19.646,A -90.000,B 90.000,C 0.000} C_DIS
LIN {X -102.968,Y -3.308,Z -19.602,A -90.000,B 90.000,C 0.000} C_DIS
LIN {X -102.934,Y -3.308,Z -19.596,A -90.000,B 90.000,C 0.000} C_DIS
LIN {X -102.772,Y -3.308,Z -19.553,A -90.000,B 90.000,C 0.000} C_DIS
LIN {X -102.669,Y -3.308,Z -19.526,A -90.000,B 90.000,C 0.000} C_DIS
LIN {X -102.657,Y -3.308,Z -19.521,A -90.000,B 90.000,C 0.000} C_DIS
LIN {X -102.636,Y -3.308,Z -19.514,A -90.000,B 90.000,C 0.000} C_DIS
LIN {X -102.461,Y -3.308,Z -19.433,A -90.000,B 90.000,C 0.000} C_DIS
LIN {X -102.425,Y -3.308,Z -19.416,A -90.000,B 90.000,C 0.000} C_DIS
LIN {X -102.415,Y -3.308,Z -19.410,A -90.000,B 90.000,C 0.000} C_DIS
LIN {X -102.413,Y -3.308,Z -19.409,A -90.000,B 90.000,C 0.000} C_DIS
LIN {X -102.402,Y -3.308,Z -19.403,A -90.000,B 90.000,C 0.000} C_DIS
LIN {X -102.303,Y -3.308,Z -19.346,A -90.000,B 90.000,C 0.000} C_DIS
LIN {X -102.283,Y -3.308,Z -19.332,A -90.000,B 90.000,C 0.000} C_DIS
LIN {X -102.281,Y -3.308,Z -19.331,A -90.000,B 90.000,C 0.000} C_DIS
LIN {X -102.279,Y -3.308,Z -19.329,A -90.000,B 90.000,C 0.000} C_DIS
LIN {X -102.268,Y -3.308,Z -19.319,A -90.000,B 90.000,C 0.000} C_DIS
LIN {X -102.261,Y -3.308,Z -19.313,A -90.000,B 90.000,C 0.000} C_DIS
LIN {X -102.260,Y -3.308,Z -19.312,A -90.000,B 90.000,C 0.000} C_DIS
LIN {X -102.212,Y -3.308,Z -19.265,A -90.000,B 90.000,C 0.000} C_DIS
LIN {X -102.179,Y -3.308,Z -19.234,A -90.000,B 90.000,C 0.000} C_DIS
LIN {X -101.952,Y -3.308,Z -19.013,A -90.000,B 90.000,C 0.000} C_DIS
LIN {X -101.919,Y -3.308,Z -18.982,A -90.000,B 90.000,C 0.000} C_DIS
LIN {X -101.630,Y -3.308,Z -18.711,A -90.000,B 90.000,C 0.000} C_DIS
LIN {X -101.602,Y -3.308,Z -18.687,A -90.000,B 90.000,C 0.000} C_DIS
LIN {X -101.343,Y -3.308,Z -18.462,A -90.000,B 90.000,C 0.000} C_DIS
LIN {X -101.325,Y -3.308,Z -18.449,A -90.000,B 90.000,C 0.000} C_DIS
LIN {X -101.128,Y -3.308,Z -18.299,A -90.000,B 90.000,C 0.000} C_DIS
LIN {X -100.996,Y -3.308,Z -18.198,A -90.000,B 90.000,C 0.000} C_DIS
LIN {X -100.707,Y -3.308,Z -17.980,A -90.000,B 90.000,C 0.000} C_DIS
LIN {X -100.683,Y -3.308,Z -17.963,A -90.000,B 90.000,C 0.000} C_DIS
LIN {X -100.655,Y -3.308,Z -17.944,A -90.000,B 90.000,C 0.000} C_DIS
LIN {X -100.638,Y -3.308,Z -17.933,A -90.000,B 90.000,C 0.000} C_DIS
LIN {X -100.258,Y -3.308,Z -17.678,A -90.000,B 90.000,C 0.000} C_DIS
LIN {X -100.184,Y -3.308,Z -17.631,A -90.000,B 90.000,C 0.000} C_DIS
LIN {X -99.922,Y -3.308,Z -17.466,A -90.000,B 90.000,C 0.000} C_DIS
LIN {X -99.652,Y -3.308,Z -17.306,A -90.000,B 90.000,C 0.000} C_DIS
LIN {X -99.432,Y -3.308,Z -17.174,A -90.000,B 90.000,C 0.000} C_DIS
LIN {X -98.996,Y -3.308,Z -16.934,A -90.000,B 90.000,C 0.000} C_DIS
LIN {X -98.827,Y -3.308,Z -16.843,A -90.000,B 90.000,C 0.000} C_DIS
LIN {X -98.365,Y -3.308,Z -16.605,A -90.000,B 90.000,C 0.000} C_DIS
LIN {X -98.101,Y -3.308,Z -16.474,A -90.000,B 90.000,C 0.000} C_DIS
LIN {X -97.957,Y -3.308,Z -16.402,A -90.000,B 90.000,C 0.000} C_DIS
LIN {X -97.700,Y -3.308,Z -16.276,A -90.000,B 90.000,C 0.000} C_DIS
LIN {X -97.581,Y -3.308,Z -16.218,A -90.000,B 90.000,C 0.000} C_DIS
LIN {X -96.875,Y -3.308,Z -15.887,A -90.000,B 90.000,C 0.000} C_DIS
LIN {X -96.345,Y -3.308,Z -15.638,A -90.000,B 90.000,C 0.000} C_DIS
LIN {X -95.962,Y -3.308,Z -15.465,A -90.000,B 90.000,C 0.000} C_DIS
LIN {X -95.748,Y -3.308,Z -15.373,A -90.000,B 90.000,C 0.000} C_DIS
LIN {X -94.976,Y -3.308,Z -15.016,A -90.000,B 90.000,C 0.000} C_DIS
LIN {X -94.975,Y -3.308,Z -15.016,A -90.000,B 90.000,C 0.000} C_DIS
LIN {X -94.965,Y -3.308,Z -15.012,A -90.000,B 90.000,C 0.000} C_DIS
LIN {X -94.152,Y -3.308,Z -14.673,A -90.000,B 90.000,C 0.000} C_DIS
LIN {X -93.926,Y -3.308,Z -14.572,A -90.000,B 90.000,C 0.000} C_DIS
LIN {X -93.291,Y -3.308,Z -14.325,A -90.000,B 90.000,C 0.000} C_DIS
LIN {X -92.827,Y -3.308,Z -14.132,A -90.000,B 90.000,C 0.000} C_DIS
LIN {X -92.621,Y -3.308,Z -14.057,A -90.000,B 90.000,C 0.000} C_DIS
LIN {X -92.399,Y -3.308,Z -13.976,A -90.000,B 90.000,C 0.000} C_DIS
LIN {X -92.206,Y -3.308,Z -13.908,A -90.000,B 90.000,C 0.000} C_DIS
LIN {X -92.158,Y -3.308,Z -13.891,A -90.000,B 90.000,C 0.000} C_DIS
LIN {X -91.813,Y -3.308,Z -13.764,A -90.000,B 90.000,C 0.000} C_DIS
LIN {X -91.617,Y -3.308,Z -13.691,A -90.000,B 90.000,C 0.000} C_DIS
LIN {X -91.358,Y -3.308,Z -13.597,A -90.000,B 90.000,C 0.000} C_DIS
LIN {X -91.263,Y -3.308,Z -13.563,A -90.000,B 90.000,C 0.000} C_DIS
LIN {X -91.042,Y -3.308,Z -13.496,A -90.000,B 90.000,C 0.000} C_DIS
LIN {X -90.104,Y -3.308,Z -13.202,A -90.000,B 90.000,C 0.000} C_DIS
LIN {X -90.103,Y -3.308,Z -13.202,A -90.000,B 90.000,C 0.000} C_DIS
LIN {X -90.101,Y -3.308,Z -13.201,A -90.000,B 90.000,C 0.000} C_DIS
LIN {X -90.094,Y -3.308,Z -13.199,A -90.000,B 90.000,C 0.000} C_DIS
LIN {X -90.045,Y -3.308,Z -13.187,A -90.000,B 90.000,C 0.000} C_DIS
LIN {X -89.102,Y -3.308,Z -12.953,A -90.000,B 90.000,C 0.000} C_DIS
LIN {X -88.733,Y -3.308,Z -12.863,A -90.000,B 90.000,C 0.000} C_DIS
LIN {X -88.660,Y -3.308,Z -12.845,A -90.000,B 90.000,C 0.000} C_DIS
LIN {X -88.457,Y -3.308,Z -12.795,A -90.000,B 90.000,C 0.000} C_DIS
LIN {X -87.615,Y -3.308,Z -12.624,A -90.000,B 90.000,C 0.000} C_DIS
LIN {X -87.187,Y -3.308,Z -12.545,A -90.000,B 90.000,C 0.000} C_DIS
LIN {X -86.503,Y -3.308,Z -12.431,A -90.000,B 90.000,C 0.000} C_DIS
LIN {X -85.658,Y -3.308,Z -12.291,A -90.000,B 90.000,C 0.000} C_DIS
LIN {X -85.640,Y -3.308,Z -12.288,A -90.000,B 90.000,C 0.000} C_DIS
LIN {X -85.626,Y -3.308,Z -12.286,A -90.000,B 90.000,C 0.000} C_DIS
LIN {X -85.605,Y -3.308,Z -12.284,A -90.000,B 90.000,C 0.000} C_DIS
LIN {X -85.574,Y -3.308,Z -12.280,A -90.000,B 90.000,C 0.000} C_DIS
LIN {X -84.109,Y -3.308,Z -12.092,A -90.000,B 90.000,C 0.000} C_DIS
LIN {X -83.298,Y -3.308,Z -12.004,A -90.000,B 90.000,C 0.000} C_DIS
LIN {X -82.591,Y -3.308,Z -11.927,A -90.000,B 90.000,C 0.000} C_DIS
LIN {X -82.516,Y -3.308,Z -11.916,A -90.000,B 90.000,C 0.000} C_DIS
LIN {X -81.058,Y -3.308,Z -11.790,A -90.000,B 90.000,C 0.000} C_DIS
LIN {X -81.035,Y -3.308,Z -11.787,A -90.000,B 90.000,C 0.000} C_DIS
LIN {X -81.023,Y -3.308,Z -11.787,A -90.000,B 90.000,C 0.000} C_DIS
LIN {X -80.916,Y -3.308,Z -11.780,A -90.000,B 90.000,C 0.000} C_DIS
LIN {X -79.937,Y -3.308,Z -11.725,A -90.000,B 90.000,C 0.000} C_DIS
LIN {X -79.569,Y -3.308,Z -11.696,A -90.000,B 90.000,C 0.000} C_DIS
LIN {X -79.358,Y -3.308,Z -11.689,A -90.000,B 90.000,C 0.000} C_DIS
LIN {X -79.087,Y -3.308,Z -11.679,A -90.000,B 90.000,C 0.000} C_DIS
LIN {X -78.290,Y -3.308,Z -11.658,A -90.000,B 90.000,C 0.000} C_DIS
LIN {X -77.842,Y -3.308,Z -11.645,A -90.000,B 90.000,C 0.000} C_DIS
LIN {X -76.991,Y -3.308,Z -11.649,A -90.000,B 90.000,C 0.000} C_DIS
LIN {X -76.714,Y -3.308,Z -11.653,A -90.000,B 90.000,C 0.000} C_DIS
LIN {X -75.850,Y -3.308,Z -11.684,A -90.000,B 90.000,C 0.000} C_DIS
LIN {X -75.791,Y -3.308,Z -11.686,A -90.000,B 90.000,C 0.000} C_DIS
LIN {X -75.693,Y -3.308,Z -11.690,A -90.000,B 90.000,C 0.000} C_DIS
LIN {X -75.555,Y -3.308,Z -11.697,A -90.000,B 90.000,C 0.000} C_DIS
LIN {X -74.823,Y -3.308,Z -11.746,A -90.000,B 90.000,C 0.000} C_DIS
LIN {X -74.575,Y -3.308,Z -11.762,A -90.000,B 90.000,C 0.000} C_DIS
LIN {X -74.210,Y -3.308,Z -11.787,A -90.000,B 90.000,C 0.000} C_DIS
LIN {X -73.468,Y -3.308,Z -11.855,A -90.000,B 90.000,C 0.000} C_DIS
LIN {X -73.219,Y -3.308,Z -11.877,A -90.000,B 90.000,C 0.000} C_DIS
LIN {X -72.497,Y -3.308,Z -11.949,A -90.000,B 90.000,C 0.000} C_DIS
LIN {X -72.201,Y -3.308,Z -11.978,A -90.000,B 90.000,C 0.000} C_DIS
LIN {X -71.491,Y -3.308,Z -12.044,A -90.000,B 90.000,C 0.000} C_DIS
LIN {X -71.116,Y -3.308,Z -12.078,A -90.000,B 90.000,C 0.000} C_DIS
LIN {X -70.645,Y -3.308,Z -12.112,A -90.000,B 90.000,C 0.000} C_DIS
LIN {X -70.395,Y -3.308,Z -12.130,A -90.000,B 90.000,C 0.000} C_DIS
LIN {X -70.206,Y -3.308,Z -12.144,A -90.000,B 90.000,C 0.000} C_DIS
LIN {X -69.622,Y -3.308,Z -12.170,A -90.000,B 90.000,C 0.000} C_DIS
LIN {X -69.060,Y -3.308,Z -12.195,A -90.000,B 90.000,C 0.000} C_DIS
LIN {X -68.228,Y -3.308,Z -12.229,A -90.000,B 90.000,C 0.000} C_DIS
LIN {X -67.641,Y -3.308,Z -12.253,A -90.000,B 90.000,C 0.000} C_DIS
LIN {X -67.448,Y -3.308,Z -12.263,A -90.000,B 90.000,C 0.000} C_DIS
LIN {X -66.587,Y -3.308,Z -12.313,A -90.000,B 90.000,C 0.000} C_DIS
LIN {X -66.030,Y -3.308,Z -12.345,A -90.000,B 90.000,C 0.000} C_DIS
LIN {X -65.733,Y -3.308,Z -12.366,A -90.000,B 90.000,C 0.000} C_DIS
LIN {X -64.878,Y -3.308,Z -12.448,A -90.000,B 90.000,C 0.000} C_DIS
LIN {X -64.364,Y -3.308,Z -12.498,A -90.000,B 90.000,C 0.000} C_DIS
LIN {X -64.190,Y -3.308,Z -12.525,A -90.000,B 90.000,C 0.000} C_DIS
LIN {X -63.414,Y -3.308,Z -12.655,A -90.000,B 90.000,C 0.000} C_DIS
LIN {X -62.945,Y -3.308,Z -12.733,A -90.000,B 90.000,C 0.000} C_DIS
LIN {X -62.651,Y -3.308,Z -12.784,A -90.000,B 90.000,C 0.000} C_DIS
LIN {X -61.958,Y -3.308,Z -12.941,A -90.000,B 90.000,C 0.000} C_DIS
LIN {X -61.517,Y -3.308,Z -13.040,A -90.000,B 90.000,C 0.000} C_DIS
LIN {X -61.335,Y -3.308,Z -13.088,A -90.000,B 90.000,C 0.000} C_DIS
LIN {X -60.694,Y -3.308,Z -13.259,A -90.000,B 90.000,C 0.000} C_DIS
LIN {X -60.287,Y -3.308,Z -13.368,A -90.000,B 90.000,C 0.000} C_DIS
LIN {X -59.655,Y -3.308,Z -13.546,A -90.000,B 90.000,C 0.000} C_DIS
LIN {X -59.316,Y -3.308,Z -13.641,A -90.000,B 90.000,C 0.000} C_DIS
LIN {X -58.624,Y -3.308,Z -13.825,A -90.000,B 90.000,C 0.000} C_DIS
LIN {X -58.504,Y -3.308,Z -13.856,A -90.000,B 90.000,C 0.000} C_DIS
LIN {X -57.592,Y -3.308,Z -14.091,A -90.000,B 90.000,C 0.000} C_DIS
LIN {X -57.590,Y -3.308,Z -14.091,A -90.000,B 90.000,C 0.000} C_DIS
LIN {X -57.588,Y -3.308,Z -14.092,A -90.000,B 90.000,C 0.000} C_DIS
LIN {X -57.524,Y -3.308,Z -14.108,A -90.000,B 90.000,C 0.000} C_DIS
LIN {X -57.125,Y -3.308,Z -14.212,A -90.000,B 90.000,C 0.000} C_DIS
LIN {X -56.513,Y -3.308,Z -14.373,A -90.000,B 90.000,C 0.000} C_DIS
LIN {X -56.481,Y -3.308,Z -14.382,A -90.000,B 90.000,C 0.000} C_DIS
LIN {X -55.391,Y -3.308,Z -14.679,A -90.000,B 90.000,C 0.000} C_DIS
LIN {X -55.318,Y -3.308,Z -14.699,A -90.000,B 90.000,C 0.000} C_DIS
LIN {X -54.883,Y -3.308,Z -14.823,A -90.000,B 90.000,C 0.000} C_DIS
LIN {X -54.866,Y -3.308,Z -14.828,A -90.000,B 90.000,C 0.000} C_DIS
LIN {X -54.854,Y -3.308,Z -14.831,A -90.000,B 90.000,C 0.000} C_DIS
LIN {X -54.813,Y -3.308,Z -14.843,A -90.000,B 90.000,C 0.000} C_DIS
LIN {X -54.808,Y -3.308,Z -14.845,A -90.000,B 90.000,C 0.000} C_DIS
LIN {X -53.975,Y -3.308,Z -15.080,A -90.000,B 90.000,C 0.000} C_DIS
LIN {X -53.957,Y -3.308,Z -15.085,A -90.000,B 90.000,C 0.000} C_DIS
LIN {X -53.873,Y -3.308,Z -15.108,A -90.000,B 90.000,C 0.000} C_DIS
LIN {X -52.348,Y -3.308,Z -15.531,A -90.000,B 90.000,C 0.000} C_DIS
LIN {X -52.215,Y -3.308,Z -15.565,A -90.000,B 90.000,C 0.000} C_DIS
LIN {X -50.337,Y -3.308,Z -16.059,A -90.000,B 90.000,C 0.000} C_DIS
LIN {X -50.088,Y -3.308,Z -16.115,A -90.000,B 90.000,C 0.000} C_DIS
LIN {X -47.841,Y -3.308,Z -16.665,A -90.000,B 90.000,C 0.000} C_DIS
LIN {X -47.243,Y -3.308,Z -16.780,A -90.000,B 90.000,C 0.000} C_DIS
LIN {X -47.233,Y -3.308,Z -16.782,A -90.000,B 90.000,C 0.000} C_DIS
LIN {X -47.231,Y -3.308,Z -16.783,A -90.000,B 90.000,C 0.000} C_DIS
LIN {X -46.660,Y -3.308,Z -16.904,A -90.000,B 90.000,C 0.000} C_DIS
LIN {X -46.272,Y -3.308,Z -16.986,A -90.000,B 90.000,C 0.000} C_DIS
LIN {X -44.865,Y -3.308,Z -17.298,A -90.000,B 90.000,C 0.000} C_DIS
LIN {X -42.380,Y -3.308,Z -17.741,A -90.000,B 90.000,C 0.000} C_DIS
LIN {X -41.422,Y -3.308,Z -17.940,A -90.000,B 90.000,C 0.000} C_DIS
LIN {X -38.142,Y -3.308,Z -18.504,A -90.000,B 90.000,C 0.000} C_DIS
LIN {X -38.084,Y -3.308,Z -18.514,A -90.000,B 90.000,C 0.000} C_DIS
LIN {X -37.902,Y -3.308,Z -18.546,A -90.000,B 90.000,C 0.000} C_DIS
LIN {X -37.347,Y -3.308,Z -18.641,A -90.000,B 90.000,C 0.000} C_DIS
LIN {X -37.170,Y -3.308,Z -18.672,A -90.000,B 90.000,C 0.000} C_DIS
LIN {X -34.585,Y -3.308,Z -19.130,A -90.000,B 90.000,C 0.000} C_DIS
LIN {X -33.319,Y -3.308,Z -19.359,A -90.000,B 90.000,C 0.000} C_DIS
LIN {X -31.564,Y -3.308,Z -19.703,A -90.000,B 90.000,C 0.000} C_DIS
LIN {X -30.017,Y -3.308,Z -20.018,A -90.000,B 90.000,C 0.000} C_DIS
LIN {X -28.859,Y -3.308,Z -20.265,A -90.000,B 90.000,C 0.000} C_DIS
LIN {X -27.094,Y -3.308,Z -20.658,A -90.000,B 90.000,C 0.000} C_DIS
LIN {X -26.383,Y -3.308,Z -20.820,A -90.000,B 90.000,C 0.000} C_DIS
LIN {X -24.408,Y -3.308,Z -21.281,A -90.000,B 90.000,C 0.000} C_DIS
LIN {X -24.050,Y -3.308,Z -21.366,A -90.000,B 90.000,C 0.000} C_DIS
LIN {X -23.989,Y -3.308,Z -21.380,A -90.000,B 90.000,C 0.000} C_DIS
LIN {X -23.761,Y -3.308,Z -21.434,A -90.000,B 90.000,C 0.000} C_DIS
LIN {X -22.172,Y -3.308,Z -21.803,A -90.000,B 90.000,C 0.000} C_DIS
LIN {X -21.772,Y -3.308,Z -21.896,A -90.000,B 90.000,C 0.000} C_DIS
LIN {X -21.771,Y -3.308,Z -21.896,A -90.000,B 90.000,C 0.000} C_DIS
LIN {X -21.762,Y -3.308,Z -21.899,A -90.000,B 90.000,C 0.000} C_DIS
LIN {X -21.683,Y -3.308,Z -21.917,A -90.000,B 90.000,C 0.000} C_DIS
LIN {X -21.341,Y -3.308,Z -21.998,A -90.000,B 90.000,C 0.000} C_DIS
LIN {X -21.256,Y -3.308,Z -22.018,A -90.000,B 90.000,C 0.000} C_DIS
LIN {X -20.886,Y -3.308,Z -22.106,A -90.000,B 90.000,C 0.000} C_DIS
LIN {X -19.135,Y -3.308,Z -22.531,A -90.000,B 90.000,C 0.000} C_DIS
LIN {X -17.521,Y -3.308,Z -22.935,A -90.000,B 90.000,C 0.000} C_DIS
LIN {X -16.888,Y -3.308,Z -23.093,A -90.000,B 90.000,C 0.000} C_DIS
LIN {X -16.242,Y -3.308,Z -23.261,A -90.000,B 90.000,C 0.000} C_DIS
LIN {X -16.118,Y -3.308,Z -23.294,A -90.000,B 90.000,C 0.000} C_DIS
LIN {X -15.781,Y -3.308,Z -23.383,A -90.000,B 90.000,C 0.000} C_DIS
LIN {X -13.901,Y -3.308,Z -23.891,A -90.000,B 90.000,C 0.000} C_DIS
LIN {X -11.822,Y -3.308,Z -24.474,A -90.000,B 90.000,C 0.000} C_DIS
LIN {X -11.144,Y -3.308,Z -24.670,A -90.000,B 90.000,C 0.000} C_DIS
LIN {X -11.073,Y -3.308,Z -24.690,A -90.000,B 90.000,C 0.000} C_DIS
LIN {X -10.704,Y -3.308,Z -24.794,A -90.000,B 90.000,C 0.000} C_DIS
LIN {X -10.644,Y -3.308,Z -24.811,A -90.000,B 90.000,C 0.000} C_DIS
LIN {X -8.913,Y -3.308,Z -25.300,A -90.000,B 90.000,C 0.000} C_DIS
LIN {X -8.903,Y -3.308,Z -25.303,A -90.000,B 90.000,C 0.000} C_DIS
LIN {X -8.526,Y -3.308,Z -25.409,A -90.000,B 90.000,C 0.000} C_DIS
LIN {X -8.474,Y -3.308,Z -25.424,A -90.000,B 90.000,C 0.000} C_DIS
LIN {X -8.449,Y -3.308,Z -25.431,A -90.000,B 90.000,C 0.000} C_DIS
LIN {X -8.139,Y -3.308,Z -25.523,A -90.000,B 90.000,C 0.000} C_DIS
LIN {X -6.359,Y -3.308,Z -26.012,A -90.000,B 90.000,C 0.000} C_DIS
LIN {X -6.065,Y -3.308,Z -26.095,A -90.000,B 90.000,C 0.000} C_DIS
LIN {X -6.054,Y -3.308,Z -26.098,A -90.000,B 90.000,C 0.000} C_DIS
LIN {X -6.012,Y -3.308,Z -26.110,A -90.000,B 90.000,C 0.000} C_DIS
LIN {X -5.895,Y -3.308,Z -26.143,A -90.000,B 90.000,C 0.000} C_DIS
LIN {X -5.206,Y -3.308,Z -26.341,A -90.000,B 90.000,C 0.000} C_DIS
LIN {X -3.778,Y -3.308,Z -26.711,A -90.000,B 90.000,C 0.000} C_DIS
LIN {X -2.131,Y -3.308,Z -27.157,A -90.000,B 90.000,C 0.000} C_DIS
LIN {X 0.360,Y -3.308,Z -27.754,A -90.000,B 90.000,C 0.000} C_DIS
LIN {X 0.926,Y -3.308,Z -27.886,A -90.000,B 90.000,C 0.000} C_DIS
LIN {X 2.625,Y -3.308,Z -28.259,A -90.000,B 90.000,C 0.000} C_DIS
LIN {X 3.825,Y -3.308,Z -28.526,A -90.000,B 90.000,C 0.000} C_DIS
LIN {X 5.944,Y -3.308,Z -28.969,A -90.000,B 90.000,C 0.000} C_DIS
LIN {X 6.499,Y -3.308,Z -29.094,A -90.000,B 90.000,C 0.000} C_DIS
LIN {X 8.503,Y -3.308,Z -29.542,A -90.000,B 90.000,C 0.000} C_DIS
LIN {X 8.864,Y -3.308,Z -29.623,A -90.000,B 90.000,C 0.000} C_DIS
LIN {X 8.951,Y -3.308,Z -29.643,A -90.000,B 90.000,C 0.000} C_DIS
LIN {X 10.880,Y -3.308,Z -30.117,A -90.000,B 90.000,C 0.000} C_DIS
LIN {X 10.884,Y -3.308,Z -30.118,A -90.000,B 90.000,C 0.000} C_DIS
LIN {X 11.039,Y -3.308,Z -30.156,A -90.000,B 90.000,C 0.000} C_DIS
LIN {X 11.449,Y -3.308,Z -30.258,A -90.000,B 90.000,C 0.000} C_DIS
LIN {X 12.620,Y -3.308,Z -30.554,A -90.000,B 90.000,C 0.000} C_DIS
LIN {X 13.678,Y -3.308,Z -30.787,A -90.000,B 90.000,C 0.000} C_DIS
LIN {X 14.213,Y -3.308,Z -30.919,A -90.000,B 90.000,C 0.000} C_DIS
LIN {X 15.733,Y -3.308,Z -31.249,A -90.000,B 90.000,C 0.000} C_DIS
LIN {X 15.744,Y -3.308,Z -31.252,A -90.000,B 90.000,C 0.000} C_DIS
LIN {X 15.766,Y -3.308,Z -31.256,A -90.000,B 90.000,C 0.000} C_DIS
LIN {X 15.914,Y -3.308,Z -31.290,A -90.000,B 90.000,C 0.000} C_DIS
LIN {X 17.430,Y -3.308,Z -31.645,A -90.000,B 90.000,C 0.000} C_DIS
LIN {X 17.433,Y -3.308,Z -31.646,A -90.000,B 90.000,C 0.000} C_DIS
LIN {X 17.541,Y -3.308,Z -31.671,A -90.000,B 90.000,C 0.000} C_DIS
LIN {X 19.125,Y -3.308,Z -32.043,A -90.000,B 90.000,C 0.000} C_DIS
LIN {X 19.131,Y -3.308,Z -32.045,A -90.000,B 90.000,C 0.000} C_DIS
LIN {X 19.329,Y -3.308,Z -32.085,A -90.000,B 90.000,C 0.000} C_DIS
LIN {X 20.821,Y -3.308,Z -32.391,A -90.000,B 90.000,C 0.000} C_DIS
LIN {X 20.841,Y -3.308,Z -32.395,A -90.000,B 90.000,C 0.000} C_DIS
LIN {X 21.375,Y -3.308,Z -32.497,A -90.000,B 90.000,C 0.000} C_DIS
LIN {X 22.389,Y -3.308,Z -32.692,A -90.000,B 90.000,C 0.000} C_DIS
LIN {X 22.409,Y -3.308,Z -32.695,A -90.000,B 90.000,C 0.000} C_DIS
LIN {X 22.942,Y -3.308,Z -32.798,A -90.000,B 90.000,C 0.000} C_DIS
LIN {X 23.854,Y -3.308,Z -32.973,A -90.000,B 90.000,C 0.000} C_DIS
LIN {X 23.876,Y -3.308,Z -32.978,A -90.000,B 90.000,C 0.000} C_DIS
LIN {X 24.429,Y -3.308,Z -33.091,A -90.000,B 90.000,C 0.000} C_DIS
LIN {X 25.280,Y -3.308,Z -33.266,A -90.000,B 90.000,C 0.000} C_DIS
LIN {X 25.305,Y -3.308,Z -33.271,A -90.000,B 90.000,C 0.000} C_DIS
LIN {X 25.905,Y -3.308,Z -33.408,A -90.000,B 90.000,C 0.000} C_DIS
LIN {X 26.733,Y -3.308,Z -33.598,A -90.000,B 90.000,C 0.000} C_DIS
LIN {X 26.763,Y -3.308,Z -33.605,A -90.000,B 90.000,C 0.000} C_DIS
LIN {X 27.509,Y -3.308,Z -33.799,A -90.000,B 90.000,C 0.000} C_DIS
LIN {X 28.279,Y -3.308,Z -33.999,A -90.000,B 90.000,C 0.000} C_DIS
LIN {X 28.315,Y -3.308,Z -34.010,A -90.000,B 90.000,C 0.000} C_DIS
LIN {X 28.386,Y -3.308,Z -34.031,A -90.000,B 90.000,C 0.000} C_DIS
LIN {X 28.466,Y -3.308,Z -34.054,A -90.000,B 90.000,C 0.000} C_DIS
LIN {X 29.162,Y -3.308,Z -34.259,A -90.000,B 90.000,C 0.000} C_DIS
LIN {X 29.981,Y -3.308,Z -34.499,A -90.000,B 90.000,C 0.000} C_DIS
LIN {X 29.992,Y -3.308,Z -34.502,A -90.000,B 90.000,C 0.000} C_DIS
LIN {X 30.141,Y -3.308,Z -34.547,A -90.000,B 90.000,C 0.000} C_DIS
LIN {X 30.199,Y -3.308,Z -34.564,A -90.000,B 90.000,C 0.000} C_DIS
LIN {X 30.339,Y -3.308,Z -34.606,A -90.000,B 90.000,C 0.000} C_DIS
LIN {X 30.448,Y -3.308,Z -34.638,A -90.000,B 90.000,C 0.000} C_DIS
LIN {X 30.492,Y -3.308,Z -34.652,A -90.000,B 90.000,C 0.000} C_DIS
LIN {X 30.606,Y -3.308,Z -34.689,A -90.000,B 90.000,C 0.000} C_DIS
LIN {X 31.622,Y -3.308,Z -35.012,A -90.000,B 90.000,C 0.000} C_DIS
LIN {X 32.046,Y -3.308,Z -35.147,A -90.000,B 90.000,C 0.000} C_DIS
LIN {X 32.165,Y -3.308,Z -35.184,A -90.000,B 90.000,C 0.000} C_DIS
LIN {X 32.311,Y -3.308,Z -35.231,A -90.000,B 90.000,C 0.000} C_DIS
LIN {X 32.365,Y -3.308,Z -35.249,A -90.000,B 90.000,C 0.000} C_DIS
LIN {X 32.409,Y -3.308,Z -35.263,A -90.000,B 90.000,C 0.000} C_DIS
LIN {X 32.934,Y -3.308,Z -35.439,A -90.000,B 90.000,C 0.000} C_DIS
LIN {X 33.241,Y -3.308,Z -35.542,A -90.000,B 90.000,C 0.000} C_DIS
LIN {X 33.980,Y -3.308,Z -35.790,A -90.000,B 90.000,C 0.000} C_DIS
LIN {X 34.020,Y -3.308,Z -35.802,A -90.000,B 90.000,C 0.000} C_DIS
LIN {X 34.326,Y -3.308,Z -35.898,A -90.000,B 90.000,C 0.000} C_DIS
LIN {X 34.359,Y -3.308,Z -35.909,A -90.000,B 90.000,C 0.000} C_DIS
LIN {X 34.412,Y -3.308,Z -35.926,A -90.000,B 90.000,C 0.000} C_DIS
LIN {X 34.738,Y -3.308,Z -36.030,A -90.000,B 90.000,C 0.000} C_DIS
LIN {X 35.817,Y -3.308,Z -36.376,A -90.000,B 90.000,C 0.000} C_DIS
LIN {X 36.236,Y -3.308,Z -36.510,A -90.000,B 90.000,C 0.000} C_DIS
LIN {X 36.487,Y -3.308,Z -36.590,A -90.000,B 90.000,C 0.000} C_DIS
LIN {X 36.549,Y -3.308,Z -36.610,A -90.000,B 90.000,C 0.000} C_DIS
LIN {X 36.652,Y -3.308,Z -36.643,A -90.000,B 90.000,C 0.000} C_DIS
LIN {X 38.703,Y -3.308,Z -37.306,A -90.000,B 90.000,C 0.000} C_DIS
LIN {X 38.911,Y -3.308,Z -37.373,A -90.000,B 90.000,C 0.000} C_DIS
LIN {X 38.963,Y -3.308,Z -37.390,A -90.000,B 90.000,C 0.000} C_DIS
